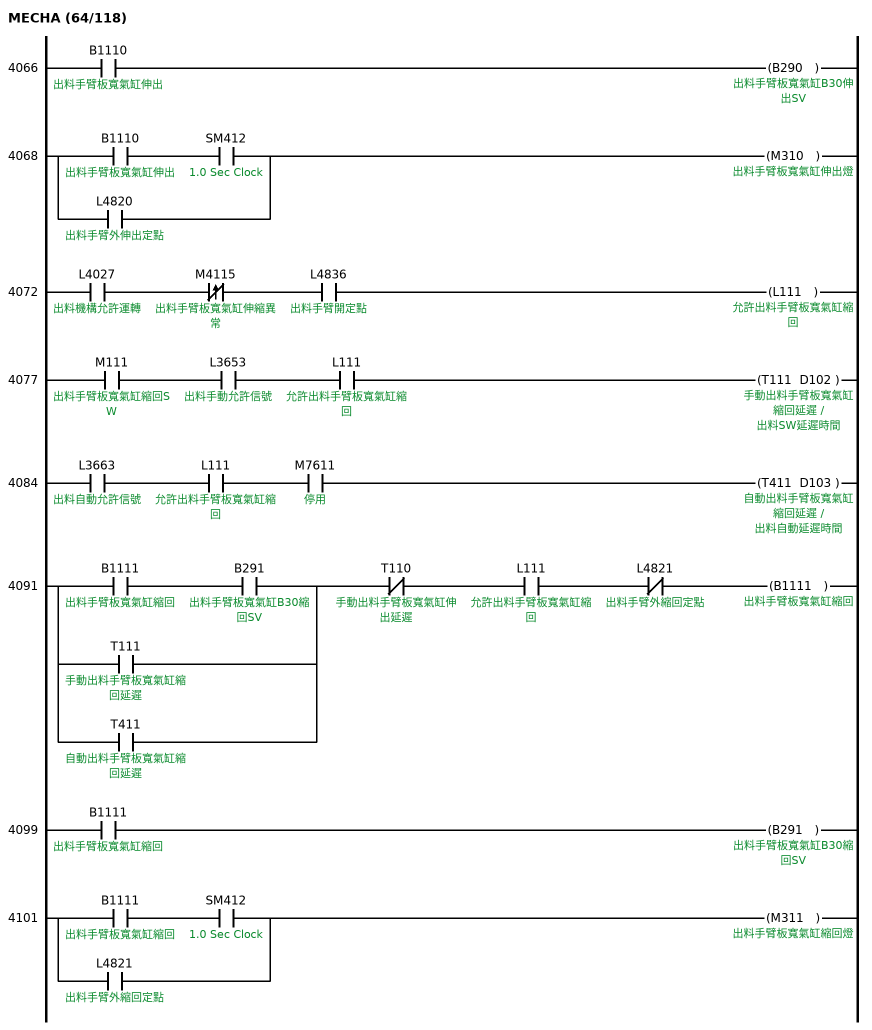
[picture p360: ladder of MECHA, rungs at steps 4066 to 4101]
4066  LD      B1110  ; 出料手臂板寬氣缸伸出
      OUT     B290  ; 出料手臂板寬氣缸B30伸出SV
4068  LD      B1110  ; 出料手臂板寬氣缸伸出
      AND     SM412  ; 1.0 Sec Clock
      OR      L4820  ; 出料手臂外伸出定點
      OUT     M310  ; 出料手臂板寬氣缸伸出燈
4072  LD      L4027  ; 出料機構允許運轉
      ANDPI   M4115  ; 出料手臂板寬氣缸伸縮異常
      AND     L4836  ; 出料手臂開定點
      OUT     L111  ; 允許出料手臂板寬氣缸縮回
4077  LD      M111  ; 出料手臂板寬氣缸縮回SW
      AND     L3653  ; 出料手動允許信號
      AND     L111  ; 允許出料手臂板寬氣缸縮回
      OUT     T111 D102  ; 手動出料手臂板寬氣缸縮回延遲 / 出料SW延遲時間
4084  LD      L3663  ; 出料自動允許信號
      AND     L111  ; 允許出料手臂板寬氣缸縮回
      AND     M7611  ; 停用
      OUT     T411 D103  ; 自動出料手臂板寬氣缸縮回延遲 / 出料自動延遲時間
4091  LD      B1111  ; 出料手臂板寬氣缸縮回
      AND     B291  ; 出料手臂板寬氣缸B30縮回SV
      OR      T111  ; 手動出料手臂板寬氣缸縮回延遲
      OR      T411  ; 自動出料手臂板寬氣缸縮回延遲
      ANI     T110  ; 手動出料手臂板寬氣缸伸出延遲
      AND     L111  ; 允許出料手臂板寬氣缸縮回
      ANI     L4821  ; 出料手臂外縮回定點
      OUT     B1111  ; 出料手臂板寬氣缸縮回
4099  LD      B1111  ; 出料手臂板寬氣缸縮回
      OUT     B291  ; 出料手臂板寬氣缸B30縮回SV
4101  LD      B1111  ; 出料手臂板寬氣缸縮回
      AND     SM412  ; 1.0 Sec Clock
      OR      L4821  ; 出料手臂外縮回定點
      OUT     M311  ; 出料手臂板寬氣缸縮回燈
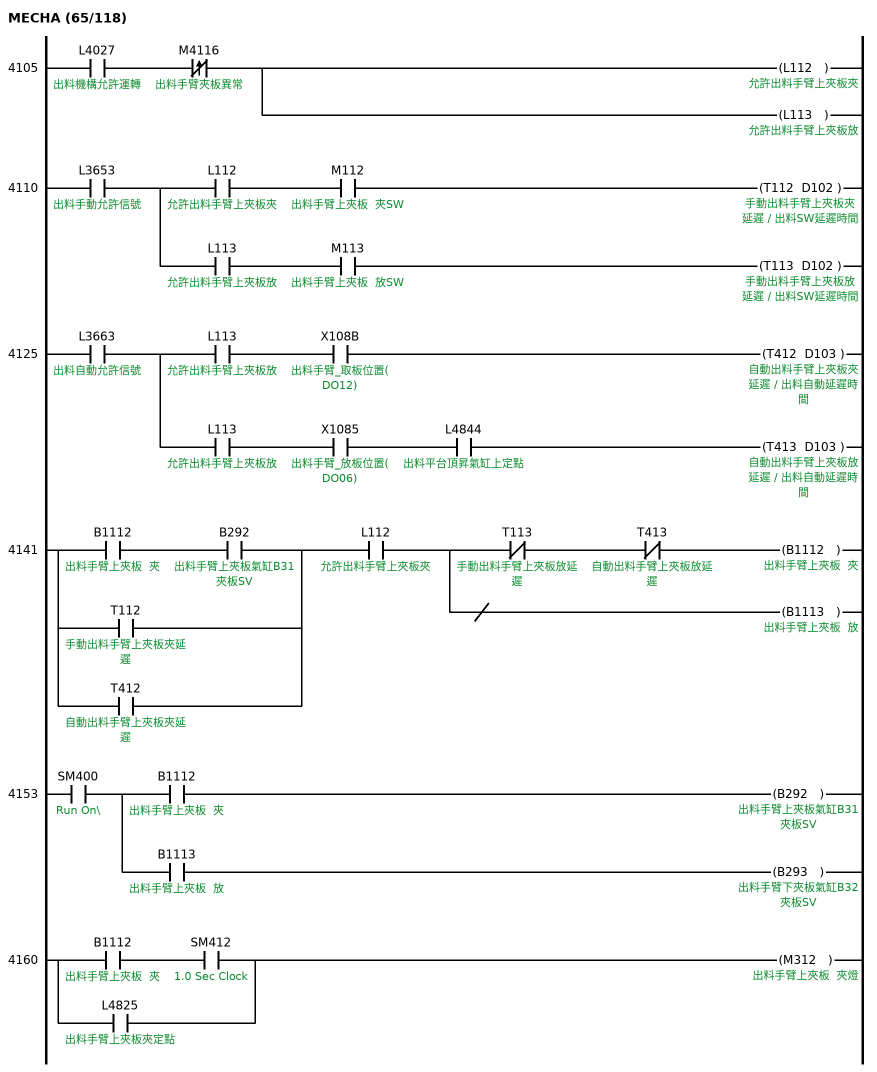
4105  LD      L4027  ; 出料機構允許運轉
      ANDPI   M4116  ; 出料手臂夾板異常
      OUT     L112  ; 允許出料手臂上夾板夾
      OUT     L113  ; 允許出料手臂上夾板放
4110  LD      L3653  ; 出料手動允許信號
      MPS
      AND     L112  ; 允許出料手臂上夾板夾
      AND     M112  ; 出料手臂上夾板  夾SW
      OUT     T112 D102  ; 手動出料手臂上夾板夾延遲 / 出料SW延遲時間
      MPP
      AND     L113  ; 允許出料手臂上夾板放
      AND     M113  ; 出料手臂上夾板  放SW
      OUT     T113 D102  ; 手動出料手臂上夾板放延遲 / 出料SW延遲時間
4125  LD      L3663  ; 出料自動允許信號
      MPS
      AND     L113  ; 允許出料手臂上夾板放
      AND     X108B  ; 出料手臂_取板位置(DO12)
      OUT     T412 D103  ; 自動出料手臂上夾板夾延遲 / 出料自動延遲時間
      MPP
      AND     L113  ; 允許出料手臂上夾板放
      AND     X1085  ; 出料手臂_放板位置(DO06)
      AND     L4844  ; 出料平台頂昇氣缸上定點
      OUT     T413 D103  ; 自動出料手臂上夾板放延遲 / 出料自動延遲時間
4141  LD      B1112  ; 出料手臂上夾板  夾
      AND     B292  ; 出料手臂上夾板氣缸B31夾板SV
      OR      T112  ; 手動出料手臂上夾板夾延遲
      OR      T412  ; 自動出料手臂上夾板夾延遲
      AND     L112  ; 允許出料手臂上夾板夾
      MPS
      ANI     T113  ; 手動出料手臂上夾板放延遲
      ANI     T413  ; 自動出料手臂上夾板放延遲
      OUT     B1112  ; 出料手臂上夾板  夾
      MPP
      INV
      OUT     B1113  ; 出料手臂上夾板  放
4153  LD      SM400  ; Run On\
      MPS
      AND     B1112  ; 出料手臂上夾板  夾
      OUT     B292  ; 出料手臂上夾板氣缸B31夾板SV
      MPP
      AND     B1113  ; 出料手臂上夾板  放
      OUT     B293  ; 出料手臂下夾板氣缸B32夾板SV
4160  LD      B1112  ; 出料手臂上夾板  夾
      AND     SM412  ; 1.0 Sec Clock
      OR      L4825  ; 出料手臂上夾板夾定點
      OUT     M312  ; 出料手臂上夾板  夾燈
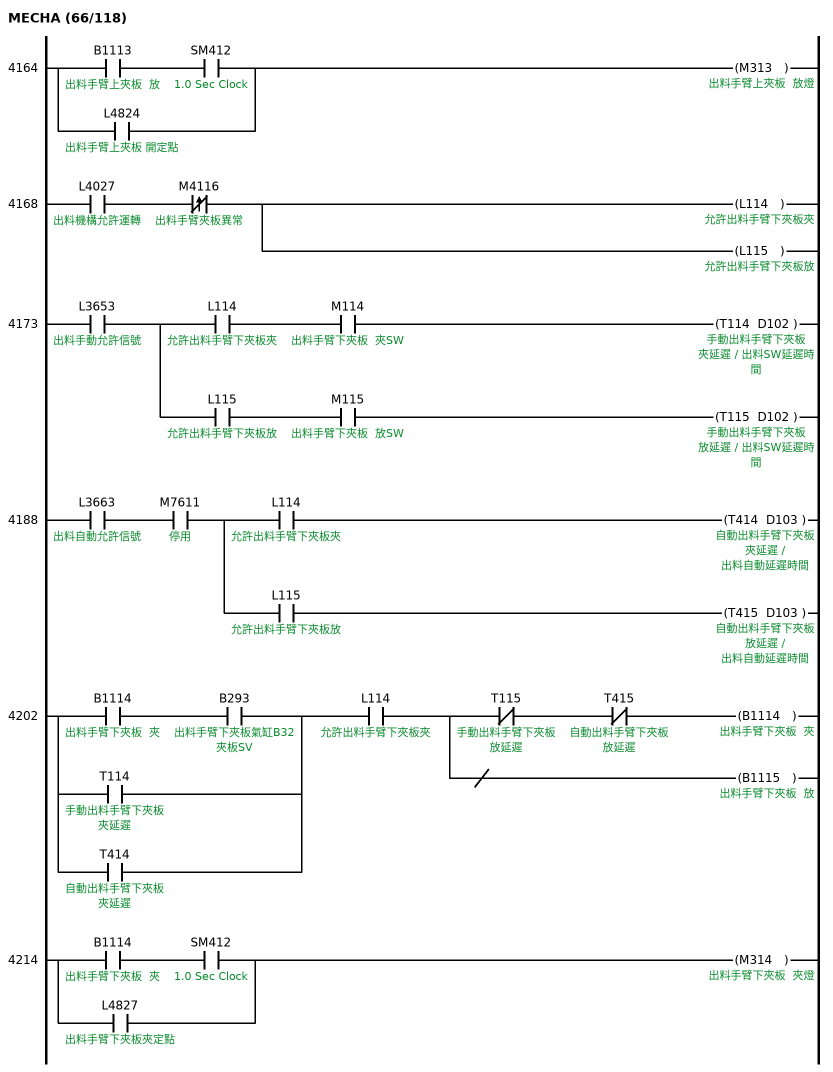
4164  LD      B1113  ; 出料手臂上夾板  放
      AND     SM412  ; 1.0 Sec Clock
      OR      L4824  ; 出料手臂上夾板 開定點
      OUT     M313  ; 出料手臂上夾板  放燈
4168  LD      L4027  ; 出料機構允許運轉
      ANDPI   M4116  ; 出料手臂夾板異常
      OUT     L114  ; 允許出料手臂下夾板夾
      OUT     L115  ; 允許出料手臂下夾板放
4173  LD      L3653  ; 出料手動允許信號
      MPS
      AND     L114  ; 允許出料手臂下夾板夾
      AND     M114  ; 出料手臂下夾板  夾SW
      OUT     T114 D102  ; 手動出料手臂下夾板  夾延遲 / 出料SW延遲時間
      MPP
      AND     L115  ; 允許出料手臂下夾板放
      AND     M115  ; 出料手臂下夾板  放SW
      OUT     T115 D102  ; 手動出料手臂下夾板  放延遲 / 出料SW延遲時間
4188  LD      L3663  ; 出料自動允許信號
      AND     M7611  ; 停用
      MPS
      AND     L114  ; 允許出料手臂下夾板夾
      OUT     T414 D103  ; 自動出料手臂下夾板  夾延遲 / 出料自動延遲時間
      MPP
      AND     L115  ; 允許出料手臂下夾板放
      OUT     T415 D103  ; 自動出料手臂下夾板  放延遲 / 出料自動延遲時間
4202  LD      B1114  ; 出料手臂下夾板  夾
      AND     B293  ; 出料手臂下夾板氣缸B32夾板SV
      OR      T114  ; 手動出料手臂下夾板  夾延遲
      OR      T414  ; 自動出料手臂下夾板  夾延遲
      AND     L114  ; 允許出料手臂下夾板夾
      MPS
      ANI     T115  ; 手動出料手臂下夾板  放延遲
      ANI     T415  ; 自動出料手臂下夾板  放延遲
      OUT     B1114  ; 出料手臂下夾板  夾
      MPP
      INV
      OUT     B1115  ; 出料手臂下夾板  放
4214  LD      B1114  ; 出料手臂下夾板  夾
      AND     SM412  ; 1.0 Sec Clock
      OR      L4827  ; 出料手臂下夾板夾定點
      OUT     M314  ; 出料手臂下夾板  夾燈
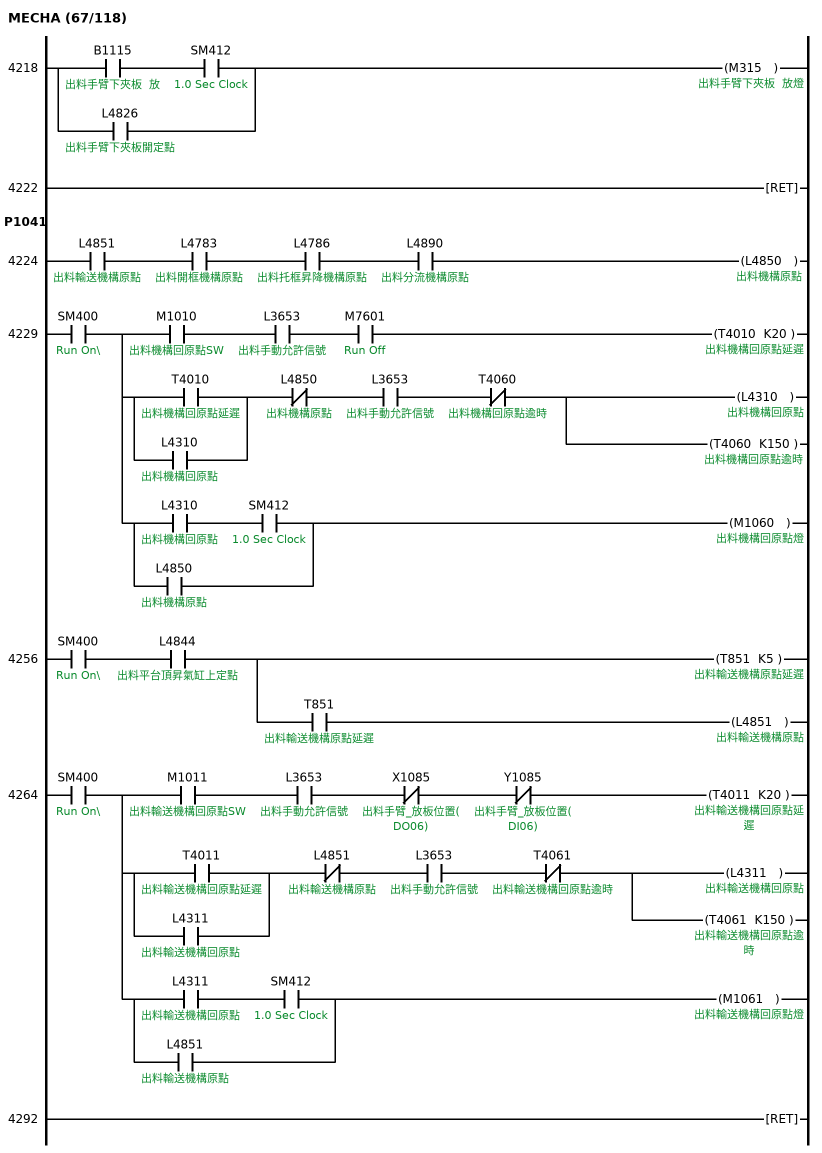
4218  LD      B1115  ; 出料手臂下夾板  放
      AND     SM412  ; 1.0 Sec Clock
      OR      L4826  ; 出料手臂下夾板開定點
      OUT     M315  ; 出料手臂下夾板  放燈
4222  RET
      P1041
4224  LD      L4851  ; 出料輸送機構原點
      AND     L4783  ; 出料開框機構原點
      AND     L4786  ; 出料托框昇降機構原點
      AND     L4890  ; 出料分流機構原點
      OUT     L4850  ; 出料機構原點
4229  LD      SM400  ; Run On\
      MPS
      AND     M1010  ; 出料機構回原點SW
      AND     L3653  ; 出料手動允許信號
      AND     M7601  ; Run Off
      OUT     T4010 K20  ; 出料機構回原點延遲
      MRD
      LD      T4010  ; 出料機構回原點延遲
      OR      L4310  ; 出料機構回原點
      ANB
      ANI     L4850  ; 出料機構原點
      AND     L3653  ; 出料手動允許信號
      ANI     T4060  ; 出料機構回原點逾時
      OUT     L4310  ; 出料機構回原點
      OUT     T4060 K150  ; 出料機構回原點逾時
      MPP
      LD      L4310  ; 出料機構回原點
      AND     SM412  ; 1.0 Sec Clock
      OR      L4850  ; 出料機構原點
      ANB
      OUT     M1060  ; 出料機構回原點燈
4256  LD      SM400  ; Run On\
      AND     L4844  ; 出料平台頂昇氣缸上定點
      OUT     T851 K5  ; 出料輸送機構原點延遲
      AND     T851  ; 出料輸送機構原點延遲
      OUT     L4851  ; 出料輸送機構原點
4264  LD      SM400  ; Run On\
      MPS
      AND     M1011  ; 出料輸送機構回原點SW
      AND     L3653  ; 出料手動允許信號
      ANI     X1085  ; 出料手臂_放板位置(DO06)
      ANI     Y1085  ; 出料手臂_放板位置(DI06)
      OUT     T4011 K20  ; 出料輸送機構回原點延遲
      MRD
      LD      T4011  ; 出料輸送機構回原點延遲
      OR      L4311  ; 出料輸送機構回原點
      ANB
      ANI     L4851  ; 出料輸送機構原點
      AND     L3653  ; 出料手動允許信號
      ANI     T4061  ; 出料輸送機構回原點逾時
      OUT     L4311  ; 出料輸送機構回原點
      OUT     T4061 K150  ; 出料輸送機構回原點逾時
      MPP
      LD      L4311  ; 出料輸送機構回原點
      AND     SM412  ; 1.0 Sec Clock
      OR      L4851  ; 出料輸送機構原點
      ANB
      OUT     M1061  ; 出料輸送機構回原點燈
4292  RET
; 出料回流下導框機構
      P1050
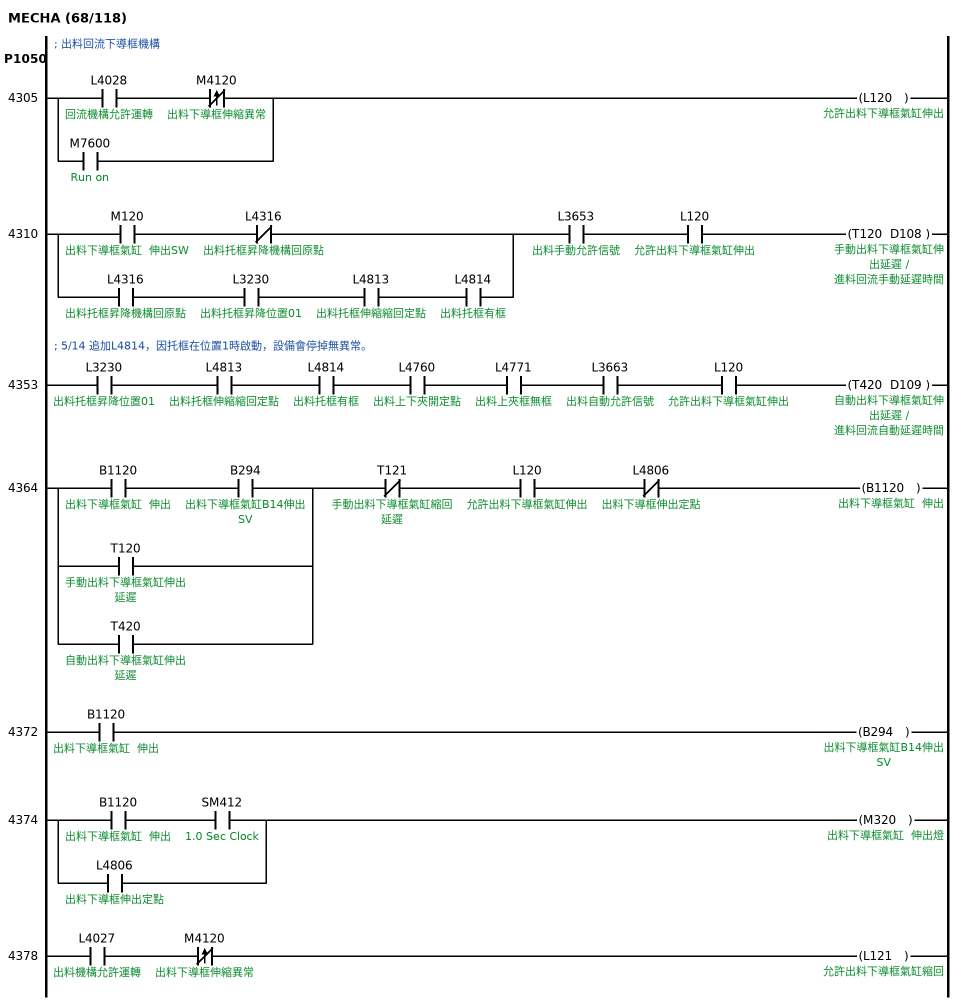
4305  LD      L4028  ; 回流機構允許運轉
      ANDPI   M4120  ; 出料下導框伸縮異常
      OR      M7600  ; Run on
      OUT     L120  ; 允許出料下導框氣缸伸出
4310  LD      M120  ; 出料下導框氣缸  伸出SW
      ANI     L4316  ; 出料托框昇降機構回原點
      LD      L4316  ; 出料托框昇降機構回原點
      AND     L3230  ; 出料托框昇降位置01
      AND     L4813  ; 出料托框伸縮縮回定點
      AND     L4814  ; 出料托框有框
      ORB
      AND     L3653  ; 出料手動允許信號
      AND     L120  ; 允許出料下導框氣缸伸出
      OUT     T120 D108  ; 手動出料下導框氣缸伸出延遲 / 進料回流手動延遲時間
; 5/14 追加L4814，因托框在位置1時啟動，設備會停掉無異常。
4353  LD      L3230  ; 出料托框昇降位置01
      AND     L4813  ; 出料托框伸縮縮回定點
      AND     L4814  ; 出料托框有框
      AND     L4760  ; 出料上下夾開定點
      AND     L4771  ; 出料上夾框無框
      AND     L3663  ; 出料自動允許信號
      AND     L120  ; 允許出料下導框氣缸伸出
      OUT     T420 D109  ; 自動出料下導框氣缸伸出延遲 / 進料回流自動延遲時間
4364  LD      B1120  ; 出料下導框氣缸  伸出
      AND     B294  ; 出料下導框氣缸B14伸出SV
      OR      T120  ; 手動出料下導框氣缸伸出延遲
      OR      T420  ; 自動出料下導框氣缸伸出延遲
      ANI     T121  ; 手動出料下導框氣缸縮回延遲
      AND     L120  ; 允許出料下導框氣缸伸出
      ANI     L4806  ; 出料下導框伸出定點
      OUT     B1120  ; 出料下導框氣缸  伸出
4372  LD      B1120  ; 出料下導框氣缸  伸出
      OUT     B294  ; 出料下導框氣缸B14伸出SV
4374  LD      B1120  ; 出料下導框氣缸  伸出
      AND     SM412  ; 1.0 Sec Clock
      OR      L4806  ; 出料下導框伸出定點
      OUT     M320  ; 出料下導框氣缸  伸出燈
4378  LD      L4027  ; 出料機構允許運轉
      ANDPI   M4120  ; 出料下導框伸縮異常
      OUT     L121  ; 允許出料下導框氣缸縮回
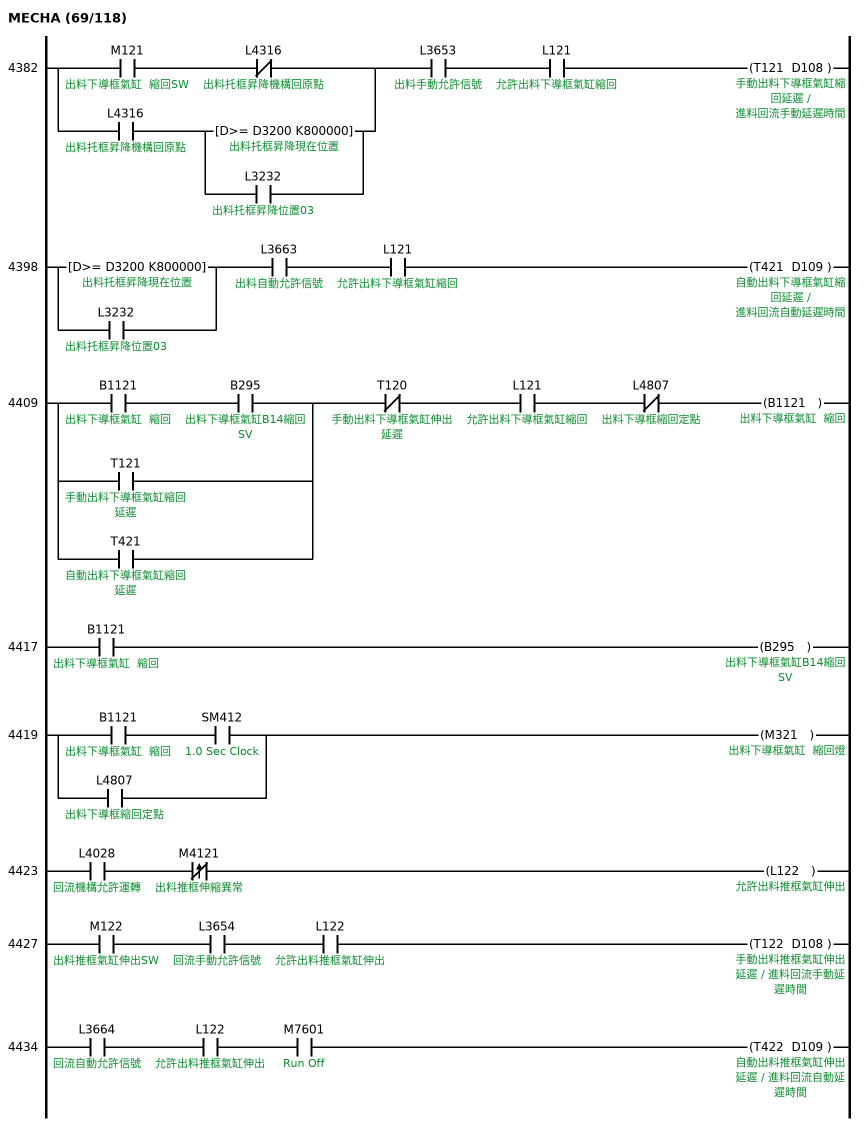
4382  LD      M121  ; 出料下導框氣缸  縮回SW
      ANI     L4316  ; 出料托框昇降機構回原點
      LD      L4316  ; 出料托框昇降機構回原點
      LDD>=   D3200 K800000  ; 出料托框昇降現在位置
      OR      L3232  ; 出料托框昇降位置03
      ANB
      ORB
      AND     L3653  ; 出料手動允許信號
      AND     L121  ; 允許出料下導框氣缸縮回
      OUT     T121 D108  ; 手動出料下導框氣缸縮回延遲 / 進料回流手動延遲時間
4398  LDD>=   D3200 K800000  ; 出料托框昇降現在位置
      OR      L3232  ; 出料托框昇降位置03
      AND     L3663  ; 出料自動允許信號
      AND     L121  ; 允許出料下導框氣缸縮回
      OUT     T421 D109  ; 自動出料下導框氣缸縮回延遲 / 進料回流自動延遲時間
4409  LD      B1121  ; 出料下導框氣缸  縮回
      AND     B295  ; 出料下導框氣缸B14縮回SV
      OR      T121  ; 手動出料下導框氣缸縮回延遲
      OR      T421  ; 自動出料下導框氣缸縮回延遲
      ANI     T120  ; 手動出料下導框氣缸伸出延遲
      AND     L121  ; 允許出料下導框氣缸縮回
      ANI     L4807  ; 出料下導框縮回定點
      OUT     B1121  ; 出料下導框氣缸  縮回
4417  LD      B1121  ; 出料下導框氣缸  縮回
      OUT     B295  ; 出料下導框氣缸B14縮回SV
4419  LD      B1121  ; 出料下導框氣缸  縮回
      AND     SM412  ; 1.0 Sec Clock
      OR      L4807  ; 出料下導框縮回定點
      OUT     M321  ; 出料下導框氣缸  縮回燈
4423  LD      L4028  ; 回流機構允許運轉
      ANDPI   M4121  ; 出料推框伸縮異常
      OUT     L122  ; 允許出料推框氣缸伸出
4427  LD      M122  ; 出料推框氣缸伸出SW
      AND     L3654  ; 回流手動允許信號
      AND     L122  ; 允許出料推框氣缸伸出
      OUT     T122 D108  ; 手動出料推框氣缸伸出延遲 / 進料回流手動延遲時間
4434  LD      L3664  ; 回流自動允許信號
      AND     L122  ; 允許出料推框氣缸伸出
      AND     M7601  ; Run Off
      OUT     T422 D109  ; 自動出料推框氣缸伸出延遲 / 進料回流自動延遲時間
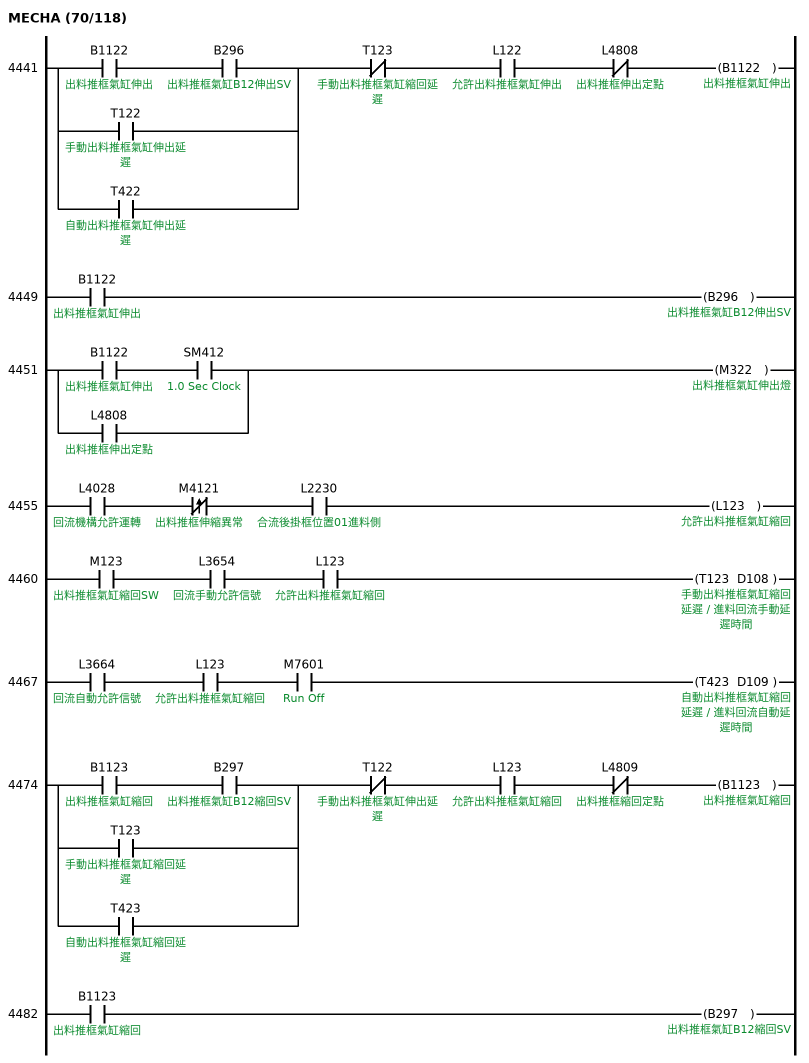
4441  LD      B1122  ; 出料推框氣缸伸出
      AND     B296  ; 出料推框氣缸B12伸出SV
      OR      T122  ; 手動出料推框氣缸伸出延遲
      OR      T422  ; 自動出料推框氣缸伸出延遲
      ANI     T123  ; 手動出料推框氣缸縮回延遲
      AND     L122  ; 允許出料推框氣缸伸出
      ANI     L4808  ; 出料推框伸出定點
      OUT     B1122  ; 出料推框氣缸伸出
4449  LD      B1122  ; 出料推框氣缸伸出
      OUT     B296  ; 出料推框氣缸B12伸出SV
4451  LD      B1122  ; 出料推框氣缸伸出
      AND     SM412  ; 1.0 Sec Clock
      OR      L4808  ; 出料推框伸出定點
      OUT     M322  ; 出料推框氣缸伸出燈
4455  LD      L4028  ; 回流機構允許運轉
      ANDPI   M4121  ; 出料推框伸縮異常
      AND     L2230  ; 合流後掛框位置01進料側
      OUT     L123  ; 允許出料推框氣缸縮回
4460  LD      M123  ; 出料推框氣缸縮回SW
      AND     L3654  ; 回流手動允許信號
      AND     L123  ; 允許出料推框氣缸縮回
      OUT     T123 D108  ; 手動出料推框氣缸縮回延遲 / 進料回流手動延遲時間
4467  LD      L3664  ; 回流自動允許信號
      AND     L123  ; 允許出料推框氣缸縮回
      AND     M7601  ; Run Off
      OUT     T423 D109  ; 自動出料推框氣缸縮回延遲 / 進料回流自動延遲時間
4474  LD      B1123  ; 出料推框氣缸縮回
      AND     B297  ; 出料推框氣缸B12縮回SV
      OR      T123  ; 手動出料推框氣缸縮回延遲
      OR      T423  ; 自動出料推框氣缸縮回延遲
      ANI     T122  ; 手動出料推框氣缸伸出延遲
      AND     L123  ; 允許出料推框氣缸縮回
      ANI     L4809  ; 出料推框縮回定點
      OUT     B1123  ; 出料推框氣缸縮回
4482  LD      B1123  ; 出料推框氣缸縮回
      OUT     B297  ; 出料推框氣缸B12縮回SV
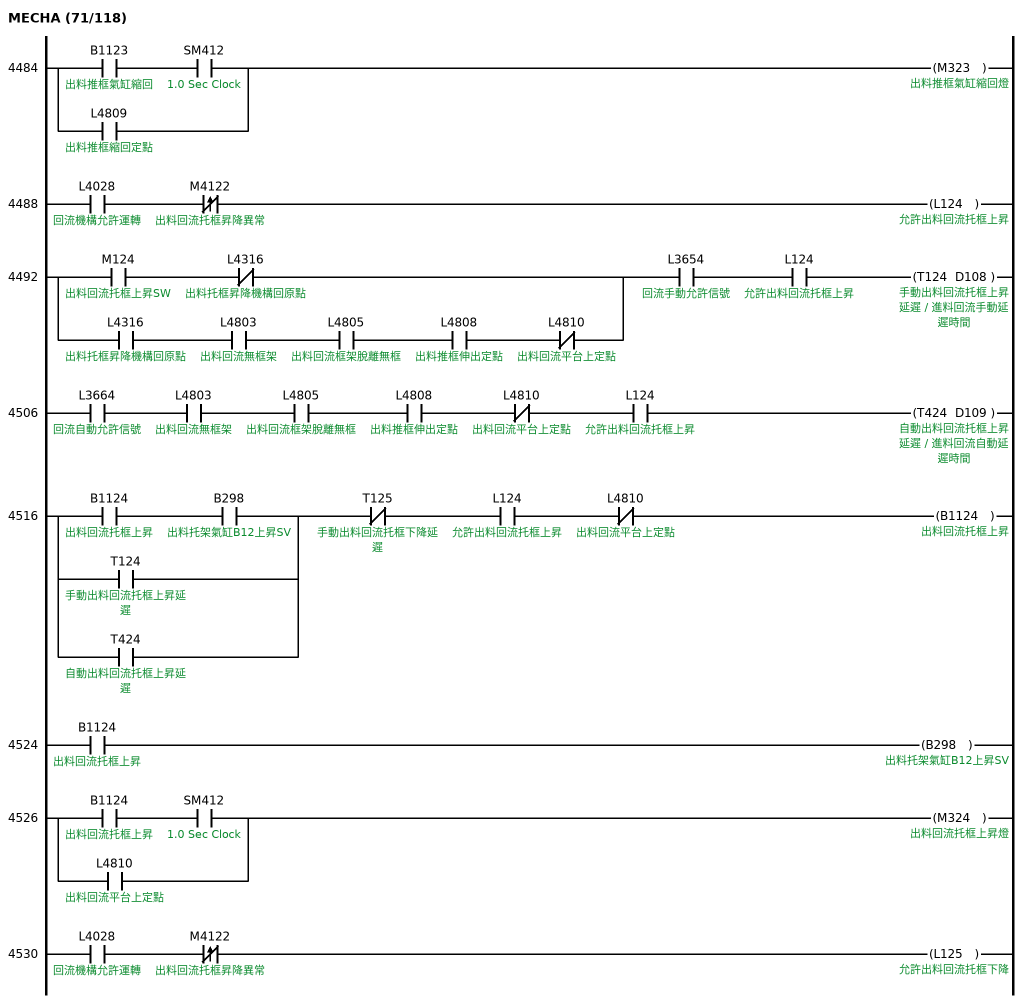
4484  LD      B1123  ; 出料推框氣缸縮回
      AND     SM412  ; 1.0 Sec Clock
      OR      L4809  ; 出料推框縮回定點
      OUT     M323  ; 出料推框氣缸縮回燈
4488  LD      L4028  ; 回流機構允許運轉
      ANDPI   M4122  ; 出料回流托框昇降異常
      OUT     L124  ; 允許出料回流托框上昇
4492  LD      M124  ; 出料回流托框上昇SW
      ANI     L4316  ; 出料托框昇降機構回原點
      LD      L4316  ; 出料托框昇降機構回原點
      AND     L4803  ; 出料回流無框架
      AND     L4805  ; 出料回流框架脫離無框
      AND     L4808  ; 出料推框伸出定點
      ANI     L4810  ; 出料回流平台上定點
      ORB
      AND     L3654  ; 回流手動允許信號
      AND     L124  ; 允許出料回流托框上昇
      OUT     T124 D108  ; 手動出料回流托框上昇延遲 / 進料回流手動延遲時間
4506  LD      L3664  ; 回流自動允許信號
      AND     L4803  ; 出料回流無框架
      AND     L4805  ; 出料回流框架脫離無框
      AND     L4808  ; 出料推框伸出定點
      ANI     L4810  ; 出料回流平台上定點
      AND     L124  ; 允許出料回流托框上昇
      OUT     T424 D109  ; 自動出料回流托框上昇延遲 / 進料回流自動延遲時間
4516  LD      B1124  ; 出料回流托框上昇
      AND     B298  ; 出料托架氣缸B12上昇SV
      OR      T124  ; 手動出料回流托框上昇延遲
      OR      T424  ; 自動出料回流托框上昇延遲
      ANI     T125  ; 手動出料回流托框下降延遲
      AND     L124  ; 允許出料回流托框上昇
      ANI     L4810  ; 出料回流平台上定點
      OUT     B1124  ; 出料回流托框上昇
4524  LD      B1124  ; 出料回流托框上昇
      OUT     B298  ; 出料托架氣缸B12上昇SV
4526  LD      B1124  ; 出料回流托框上昇
      AND     SM412  ; 1.0 Sec Clock
      OR      L4810  ; 出料回流平台上定點
      OUT     M324  ; 出料回流托框上昇燈
4530  LD      L4028  ; 回流機構允許運轉
      ANDPI   M4122  ; 出料回流托框昇降異常
      OUT     L125  ; 允許出料回流托框下降
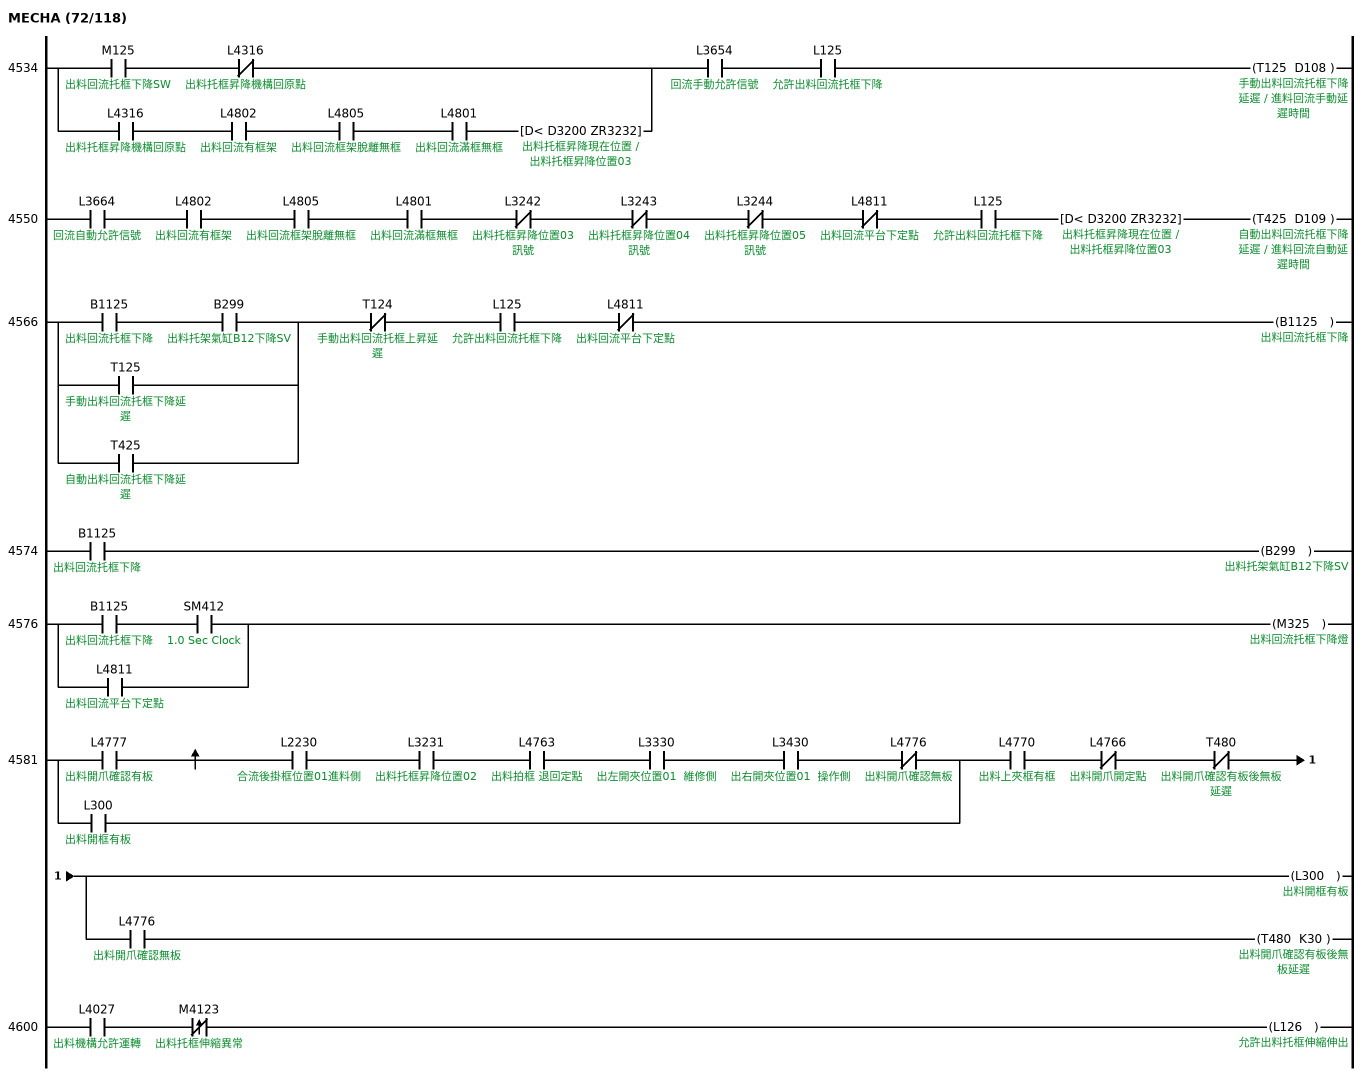
4534  LD      M125  ; 出料回流托框下降SW
      ANI     L4316  ; 出料托框昇降機構回原點
      LD      L4316  ; 出料托框昇降機構回原點
      AND     L4802  ; 出料回流有框架
      AND     L4805  ; 出料回流框架脫離無框
      AND     L4801  ; 出料回流滿框無框
      ANDD<   D3200 ZR3232  ; 出料托框昇降現在位置 / 出料托框昇降位置03
      ORB
      AND     L3654  ; 回流手動允許信號
      AND     L125  ; 允許出料回流托框下降
      OUT     T125 D108  ; 手動出料回流托框下降延遲 / 進料回流手動延遲時間
4550  LD      L3664  ; 回流自動允許信號
      AND     L4802  ; 出料回流有框架
      AND     L4805  ; 出料回流框架脫離無框
      AND     L4801  ; 出料回流滿框無框
      ANI     L3242  ; 出料托框昇降位置03 訊號
      ANI     L3243  ; 出料托框昇降位置04 訊號
      ANI     L3244  ; 出料托框昇降位置05 訊號
      ANI     L4811  ; 出料回流平台下定點
      AND     L125  ; 允許出料回流托框下降
      ANDD<   D3200 ZR3232  ; 出料托框昇降現在位置 / 出料托框昇降位置03
      OUT     T425 D109  ; 自動出料回流托框下降延遲 / 進料回流自動延遲時間
4566  LD      B1125  ; 出料回流托框下降
      AND     B299  ; 出料托架氣缸B12下降SV
      OR      T125  ; 手動出料回流托框下降延遲
      OR      T425  ; 自動出料回流托框下降延遲
      ANI     T124  ; 手動出料回流托框上昇延遲
      AND     L125  ; 允許出料回流托框下降
      ANI     L4811  ; 出料回流平台下定點
      OUT     B1125  ; 出料回流托框下降
4574  LD      B1125  ; 出料回流托框下降
      OUT     B299  ; 出料托架氣缸B12下降SV
4576  LD      B1125  ; 出料回流托框下降
      AND     SM412  ; 1.0 Sec Clock
      OR      L4811  ; 出料回流平台下定點
      OUT     M325  ; 出料回流托框下降燈
4581  LD      L4777  ; 出料開爪確認有板
      MEP
      AND     L2230  ; 合流後掛框位置01進料側
      AND     L3231  ; 出料托框昇降位置02
      AND     L4763  ; 出料拍框 退回定點
      AND     L3330  ; 出左開夾位置01  維修側
      AND     L3430  ; 出右開夾位置01  操作側
      ANI     L4776  ; 出料開爪確認無板
      OR      L300  ; 出料開框有板
      AND     L4770  ; 出料上夾框有框
      ANI     L4766  ; 出料開爪開定點
      ANI     T480  ; 出料開爪確認有板後無板延遲
      OUT     L300  ; 出料開框有板
      AND     L4776  ; 出料開爪確認無板
      OUT     T480 K30  ; 出料開爪確認有板後無板延遲
4600  LD      L4027  ; 出料機構允許運轉
      ANDPI   M4123  ; 出料托框伸縮異常
      OUT     L126  ; 允許出料托框伸縮伸出
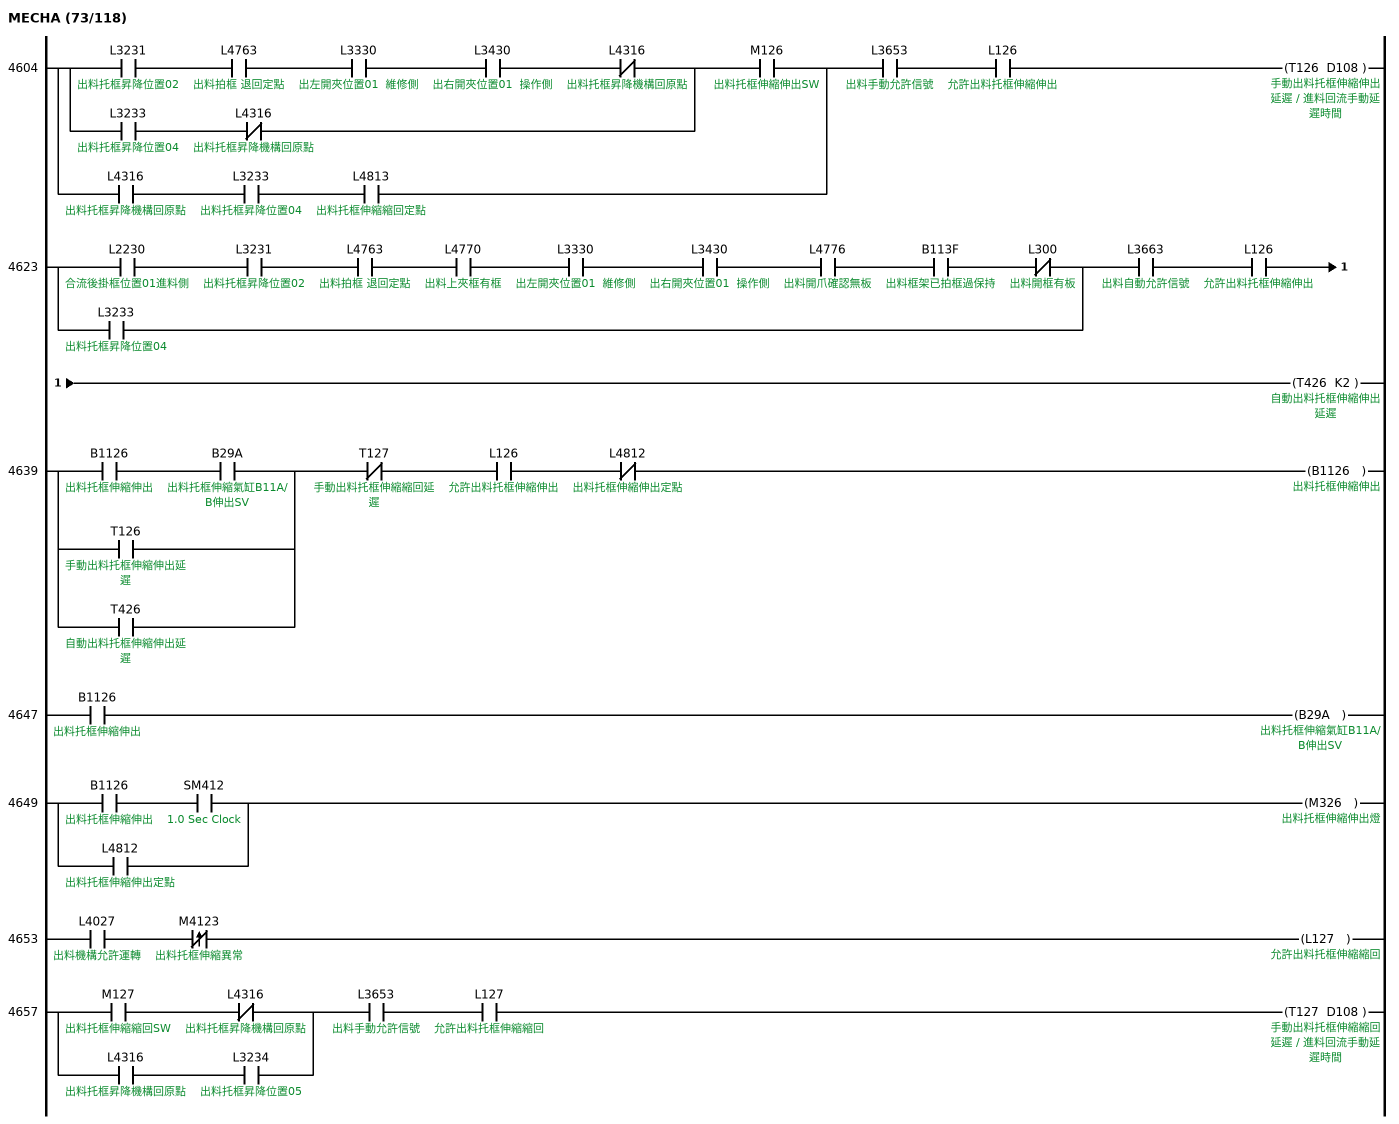
4604  LD      L3231  ; 出料托框昇降位置02
      AND     L4763  ; 出料拍框 退回定點
      AND     L3330  ; 出左開夾位置01  維修側
      AND     L3430  ; 出右開夾位置01  操作側
      ANI     L4316  ; 出料托框昇降機構回原點
      LD      L3233  ; 出料托框昇降位置04
      ANI     L4316  ; 出料托框昇降機構回原點
      ORB
      AND     M126  ; 出料托框伸縮伸出SW
      LD      L4316  ; 出料托框昇降機構回原點
      AND     L3233  ; 出料托框昇降位置04
      AND     L4813  ; 出料托框伸縮縮回定點
      ORB
      AND     L3653  ; 出料手動允許信號
      AND     L126  ; 允許出料托框伸縮伸出
      OUT     T126 D108  ; 手動出料托框伸縮伸出延遲 / 進料回流手動延遲時間
4623  LD      L2230  ; 合流後掛框位置01進料側
      AND     L3231  ; 出料托框昇降位置02
      AND     L4763  ; 出料拍框 退回定點
      AND     L4770  ; 出料上夾框有框
      AND     L3330  ; 出左開夾位置01  維修側
      AND     L3430  ; 出右開夾位置01  操作側
      AND     L4776  ; 出料開爪確認無板
      AND     B113F  ; 出料框架已拍框過保持
      ANI     L300  ; 出料開框有板
      OR      L3233  ; 出料托框昇降位置04
      AND     L3663  ; 出料自動允許信號
      AND     L126  ; 允許出料托框伸縮伸出
      OUT     T426 K2  ; 自動出料托框伸縮伸出延遲
4639  LD      B1126  ; 出料托框伸縮伸出
      AND     B29A  ; 出料托框伸縮氣缸B11A/B伸出SV
      OR      T126  ; 手動出料托框伸縮伸出延遲
      OR      T426  ; 自動出料托框伸縮伸出延遲
      ANI     T127  ; 手動出料托框伸縮縮回延遲
      AND     L126  ; 允許出料托框伸縮伸出
      ANI     L4812  ; 出料托框伸縮伸出定點
      OUT     B1126  ; 出料托框伸縮伸出
4647  LD      B1126  ; 出料托框伸縮伸出
      OUT     B29A  ; 出料托框伸縮氣缸B11A/B伸出SV
4649  LD      B1126  ; 出料托框伸縮伸出
      AND     SM412  ; 1.0 Sec Clock
      OR      L4812  ; 出料托框伸縮伸出定點
      OUT     M326  ; 出料托框伸縮伸出燈
4653  LD      L4027  ; 出料機構允許運轉
      ANDPI   M4123  ; 出料托框伸縮異常
      OUT     L127  ; 允許出料托框伸縮縮回
4657  LD      M127  ; 出料托框伸縮縮回SW
      ANI     L4316  ; 出料托框昇降機構回原點
      LD      L4316  ; 出料托框昇降機構回原點
      AND     L3234  ; 出料托框昇降位置05
      ORB
      AND     L3653  ; 出料手動允許信號
      AND     L127  ; 允許出料托框伸縮縮回
      OUT     T127 D108  ; 手動出料托框伸縮縮回延遲 / 進料回流手動延遲時間
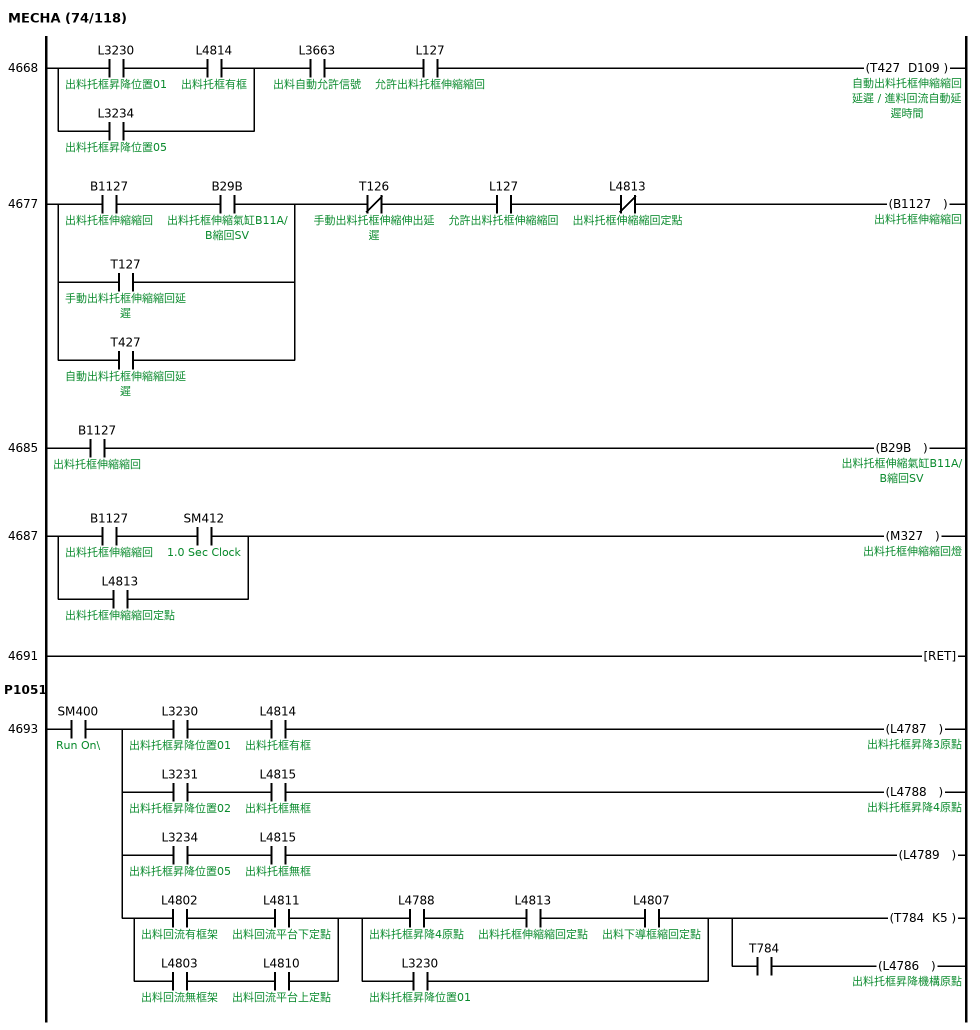
4668  LD      L3230  ; 出料托框昇降位置01
      AND     L4814  ; 出料托框有框
      OR      L3234  ; 出料托框昇降位置05
      AND     L3663  ; 出料自動允許信號
      AND     L127  ; 允許出料托框伸縮縮回
      OUT     T427 D109  ; 自動出料托框伸縮縮回延遲 / 進料回流自動延遲時間
4677  LD      B1127  ; 出料托框伸縮縮回
      AND     B29B  ; 出料托框伸縮氣缸B11A/B縮回SV
      OR      T127  ; 手動出料托框伸縮縮回延遲
      OR      T427  ; 自動出料托框伸縮縮回延遲
      ANI     T126  ; 手動出料托框伸縮伸出延遲
      AND     L127  ; 允許出料托框伸縮縮回
      ANI     L4813  ; 出料托框伸縮縮回定點
      OUT     B1127  ; 出料托框伸縮縮回
4685  LD      B1127  ; 出料托框伸縮縮回
      OUT     B29B  ; 出料托框伸縮氣缸B11A/B縮回SV
4687  LD      B1127  ; 出料托框伸縮縮回
      AND     SM412  ; 1.0 Sec Clock
      OR      L4813  ; 出料托框伸縮縮回定點
      OUT     M327  ; 出料托框伸縮縮回燈
4691  RET
      P1051
4693  LD      SM400  ; Run On\
      MPS
      AND     L3230  ; 出料托框昇降位置01
      AND     L4814  ; 出料托框有框
      OUT     L4787  ; 出料托框昇降3原點
      MRD
      AND     L3231  ; 出料托框昇降位置02
      AND     L4815  ; 出料托框無框
      OUT     L4788  ; 出料托框昇降4原點
      MRD
      AND     L3234  ; 出料托框昇降位置05
      AND     L4815  ; 出料托框無框
      OUT     L4789
      MPP
      LD      L4802  ; 出料回流有框架
      AND     L4811  ; 出料回流平台下定點
      LD      L4803  ; 出料回流無框架
      AND     L4810  ; 出料回流平台上定點
      ORB
      ANB
      LD      L4788  ; 出料托框昇降4原點
      AND     L4813  ; 出料托框伸縮縮回定點
      AND     L4807  ; 出料下導框縮回定點
      OR      L3230  ; 出料托框昇降位置01
      ANB
      OUT     T784 K5
      AND     T784
      OUT     L4786  ; 出料托框昇降機構原點
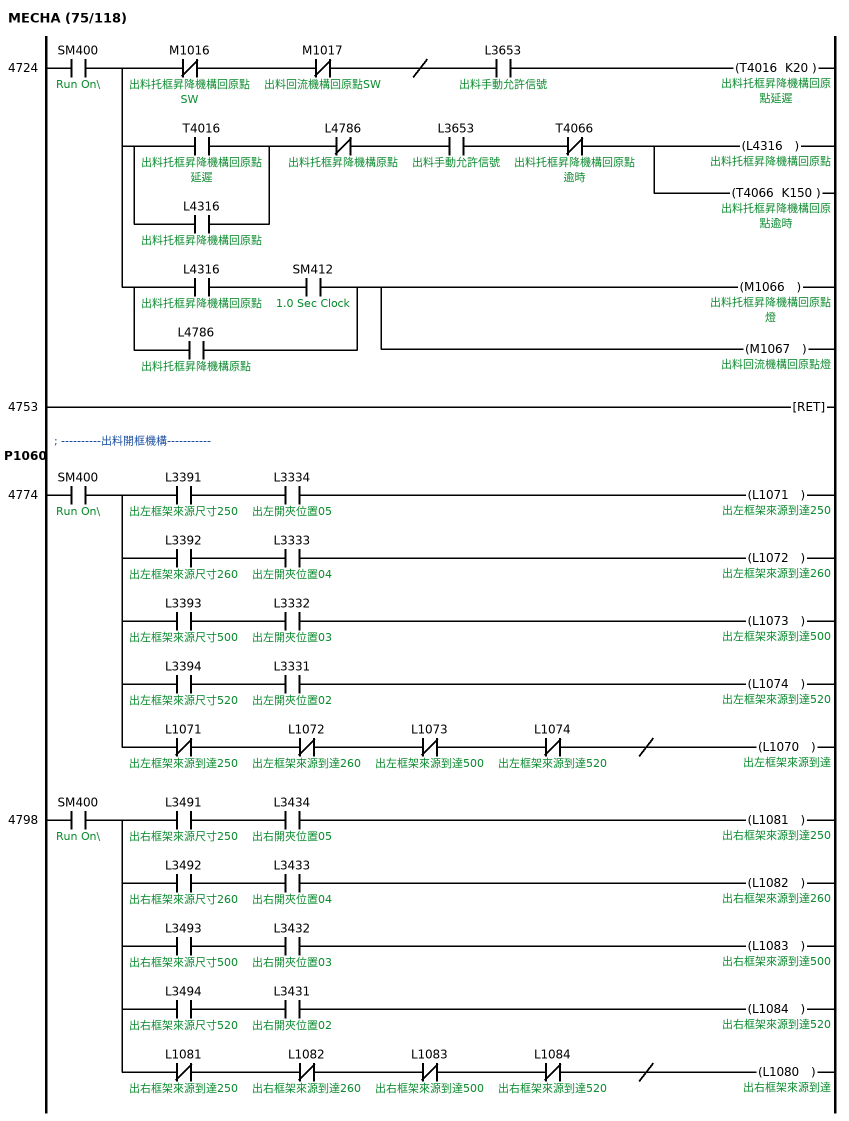
4724  LD      SM400  ; Run On\
      MPS
      ANI     M1016  ; 出料托框昇降機構回原點SW
      ANI     M1017  ; 出料回流機構回原點SW
      INV
      AND     L3653  ; 出料手動允許信號
      OUT     T4016 K20  ; 出料托框昇降機構回原點延遲
      MRD
      LD      T4016  ; 出料托框昇降機構回原點延遲
      OR      L4316  ; 出料托框昇降機構回原點
      ANB
      ANI     L4786  ; 出料托框昇降機構原點
      AND     L3653  ; 出料手動允許信號
      ANI     T4066  ; 出料托框昇降機構回原點逾時
      OUT     L4316  ; 出料托框昇降機構回原點
      OUT     T4066 K150  ; 出料托框昇降機構回原點逾時
      MPP
      LD      L4316  ; 出料托框昇降機構回原點
      AND     SM412  ; 1.0 Sec Clock
      OR      L4786  ; 出料托框昇降機構原點
      ANB
      OUT     M1066  ; 出料托框昇降機構回原點燈
      OUT     M1067  ; 出料回流機構回原點燈
4753  RET
; ----------出料開框機構-----------
      P1060
4774  LD      SM400  ; Run On\
      MPS
      AND     L3391  ; 出左框架來源尺寸250
      AND     L3334  ; 出左開夾位置05
      OUT     L1071  ; 出左框架來源到達250
      MRD
      AND     L3392  ; 出左框架來源尺寸260
      AND     L3333  ; 出左開夾位置04
      OUT     L1072  ; 出左框架來源到達260
      MRD
      AND     L3393  ; 出左框架來源尺寸500
      AND     L3332  ; 出左開夾位置03
      OUT     L1073  ; 出左框架來源到達500
      MRD
      AND     L3394  ; 出左框架來源尺寸520
      AND     L3331  ; 出左開夾位置02
      OUT     L1074  ; 出左框架來源到達520
      MPP
      ANI     L1071  ; 出左框架來源到達250
      ANI     L1072  ; 出左框架來源到達260
      ANI     L1073  ; 出左框架來源到達500
      ANI     L1074  ; 出左框架來源到達520
      INV
      OUT     L1070  ; 出左框架來源到達
4798  LD      SM400  ; Run On\
      MPS
      AND     L3491  ; 出右框架來源尺寸250
      AND     L3434  ; 出右開夾位置05
      OUT     L1081  ; 出右框架來源到達250
      MRD
      AND     L3492  ; 出右框架來源尺寸260
      AND     L3433  ; 出右開夾位置04
      OUT     L1082  ; 出右框架來源到達260
      MRD
      AND     L3493  ; 出右框架來源尺寸500
      AND     L3432  ; 出右開夾位置03
      OUT     L1083  ; 出右框架來源到達500
      MRD
      AND     L3494  ; 出右框架來源尺寸520
      AND     L3431  ; 出右開夾位置02
      OUT     L1084  ; 出右框架來源到達520
      MPP
      ANI     L1081  ; 出右框架來源到達250
      ANI     L1082  ; 出右框架來源到達260
      ANI     L1083  ; 出右框架來源到達500
      ANI     L1084  ; 出右框架來源到達520
      INV
      OUT     L1080  ; 出右框架來源到達
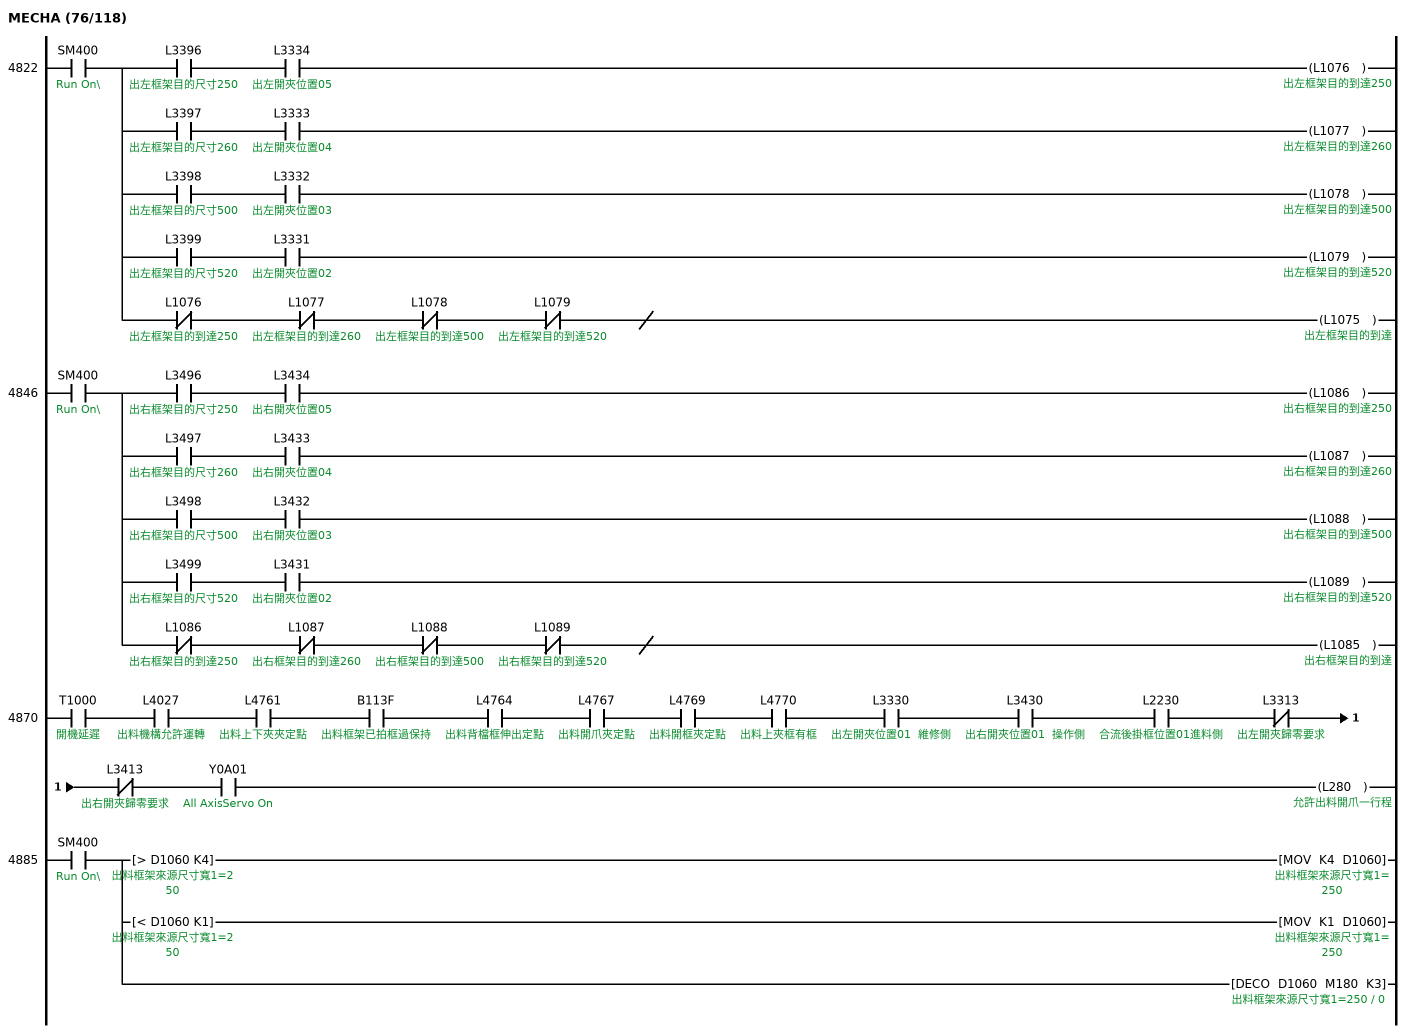
4822  LD      SM400  ; Run On\
      MPS
      AND     L3396  ; 出左框架目的尺寸250
      AND     L3334  ; 出左開夾位置05
      OUT     L1076  ; 出左框架目的到達250
      MRD
      AND     L3397  ; 出左框架目的尺寸260
      AND     L3333  ; 出左開夾位置04
      OUT     L1077  ; 出左框架目的到達260
      MRD
      AND     L3398  ; 出左框架目的尺寸500
      AND     L3332  ; 出左開夾位置03
      OUT     L1078  ; 出左框架目的到達500
      MRD
      AND     L3399  ; 出左框架目的尺寸520
      AND     L3331  ; 出左開夾位置02
      OUT     L1079  ; 出左框架目的到達520
      MPP
      ANI     L1076  ; 出左框架目的到達250
      ANI     L1077  ; 出左框架目的到達260
      ANI     L1078  ; 出左框架目的到達500
      ANI     L1079  ; 出左框架目的到達520
      INV
      OUT     L1075  ; 出左框架目的到達
4846  LD      SM400  ; Run On\
      MPS
      AND     L3496  ; 出右框架目的尺寸250
      AND     L3434  ; 出右開夾位置05
      OUT     L1086  ; 出右框架目的到達250
      MRD
      AND     L3497  ; 出右框架目的尺寸260
      AND     L3433  ; 出右開夾位置04
      OUT     L1087  ; 出右框架目的到達260
      MRD
      AND     L3498  ; 出右框架目的尺寸500
      AND     L3432  ; 出右開夾位置03
      OUT     L1088  ; 出右框架目的到達500
      MRD
      AND     L3499  ; 出右框架目的尺寸520
      AND     L3431  ; 出右開夾位置02
      OUT     L1089  ; 出右框架目的到達520
      MPP
      ANI     L1086  ; 出右框架目的到達250
      ANI     L1087  ; 出右框架目的到達260
      ANI     L1088  ; 出右框架目的到達500
      ANI     L1089  ; 出右框架目的到達520
      INV
      OUT     L1085  ; 出右框架目的到達
4870  LD      T1000  ; 開機延遲
      AND     L4027  ; 出料機構允許運轉
      AND     L4761  ; 出料上下夾夾定點
      AND     B113F  ; 出料框架已拍框過保持
      AND     L4764  ; 出料背檔框伸出定點
      AND     L4767  ; 出料開爪夾定點
      AND     L4769  ; 出料開框夾定點
      AND     L4770  ; 出料上夾框有框
      AND     L3330  ; 出左開夾位置01  維修側
      AND     L3430  ; 出右開夾位置01  操作側
      AND     L2230  ; 合流後掛框位置01進料側
      ANI     L3313  ; 出左開夾歸零要求
      ANI     L3413  ; 出右開夾歸零要求
      AND     Y0A01  ; All AxisServo On
      OUT     L280  ; 允許出料開爪一行程
4885  LD      SM400  ; Run On\
      MPS
      AND>    D1060 K4  ; 出料框架來源尺寸寬1=250
      MOV     K4 D1060
      MRD
      AND<    D1060 K1  ; 出料框架來源尺寸寬1=250
      MOV     K1 D1060
      MPP
      DECO    D1060 M180 K3  ; 0
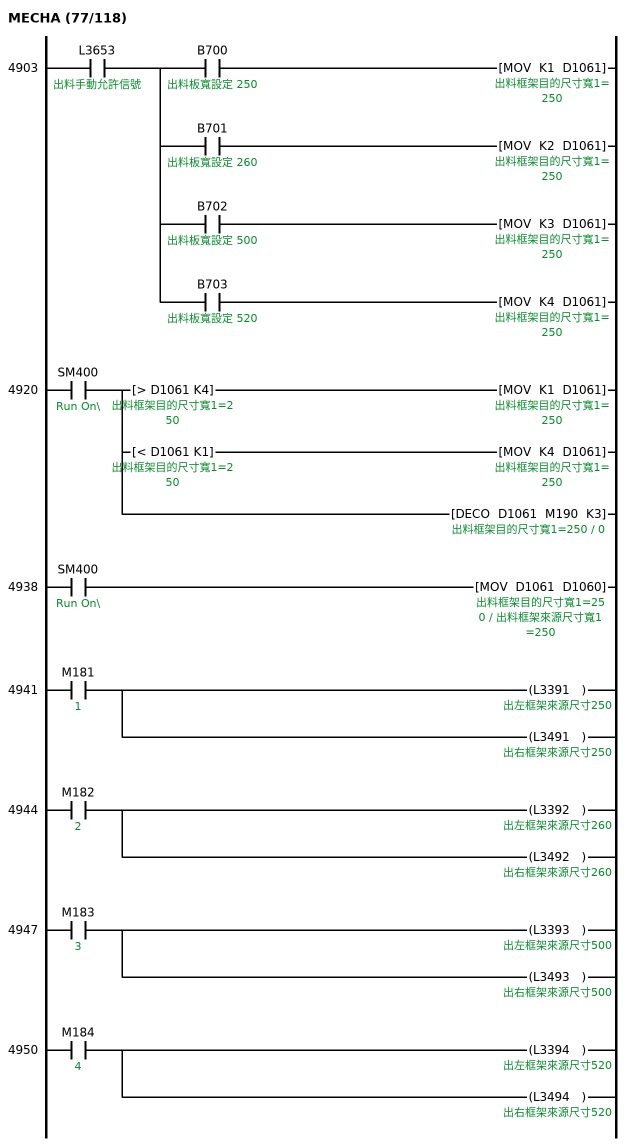
4903  LD      L3653  ; 出料手動允許信號
      MPS
      AND     B700  ; 出料板寬設定 250
      MOV     K1 D1061  ; 出料框架目的尺寸寬1=250
      MRD
      AND     B701  ; 出料板寬設定 260
      MOV     K2 D1061
      MRD
      AND     B702  ; 出料板寬設定 500
      MOV     K3 D1061
      MPP
      AND     B703  ; 出料板寬設定 520
      MOV     K4 D1061
4920  LD      SM400  ; Run On\
      MPS
      AND>    D1061 K4  ; 出料框架目的尺寸寬1=250
      MOV     K1 D1061
      MRD
      AND<    D1061 K1  ; 出料框架目的尺寸寬1=250
      MOV     K4 D1061
      MPP
      DECO    D1061 M190 K3  ; 0
4938  LD      SM400  ; Run On\
      MOV     D1061 D1060
4941  LD      M181  ; 1
      OUT     L3391  ; 出左框架來源尺寸250
      OUT     L3491  ; 出右框架來源尺寸250
4944  LD      M182  ; 2
      OUT     L3392  ; 出左框架來源尺寸260
      OUT     L3492  ; 出右框架來源尺寸260
4947  LD      M183  ; 3
      OUT     L3393  ; 出左框架來源尺寸500
      OUT     L3493  ; 出右框架來源尺寸500
4950  LD      M184  ; 4
      OUT     L3394  ; 出左框架來源尺寸520
      OUT     L3494  ; 出右框架來源尺寸520
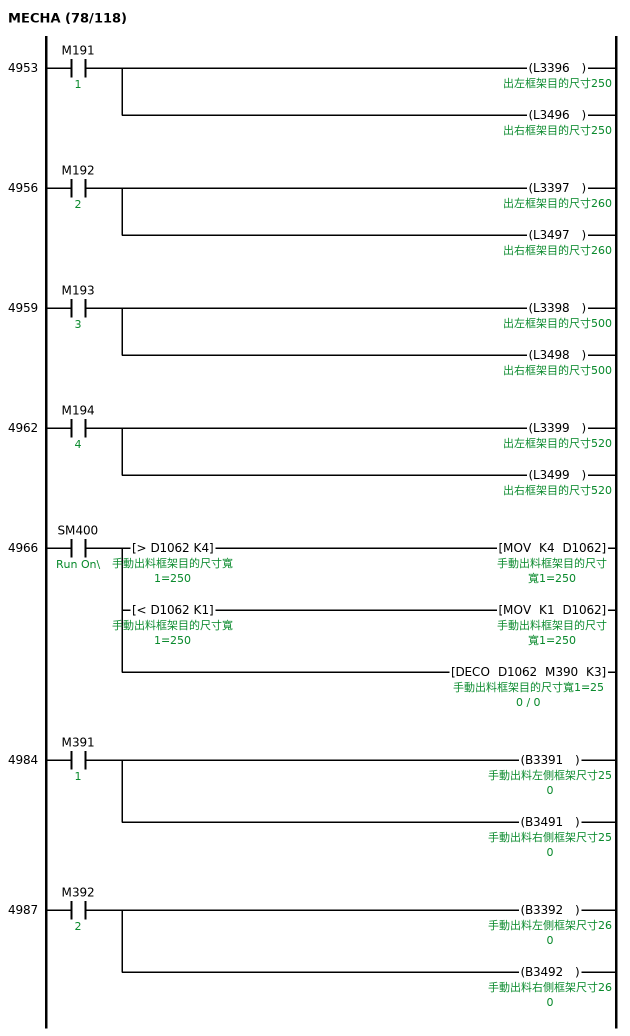
4953  LD      M191  ; 1
      OUT     L3396  ; 出左框架目的尺寸250
      OUT     L3496  ; 出右框架目的尺寸250
4956  LD      M192  ; 2
      OUT     L3397  ; 出左框架目的尺寸260
      OUT     L3497  ; 出右框架目的尺寸260
4959  LD      M193  ; 3
      OUT     L3398  ; 出左框架目的尺寸500
      OUT     L3498  ; 出右框架目的尺寸500
4962  LD      M194  ; 4
      OUT     L3399  ; 出左框架目的尺寸520
      OUT     L3499  ; 出右框架目的尺寸520
4966  LD      SM400  ; Run On\
      MPS
      AND>    D1062 K4  ; 手動出料框架目的尺寸寬1=250
      MOV     K4 D1062
      MRD
      AND<    D1062 K1  ; 手動出料框架目的尺寸寬1=250
      MOV     K1 D1062
      MPP
      DECO    D1062 M390 K3  ; 0
4984  LD      M391  ; 1
      OUT     B3391  ; 手動出料左側框架尺寸250
      OUT     B3491  ; 手動出料右側框架尺寸250
4987  LD      M392  ; 2
      OUT     B3392  ; 手動出料左側框架尺寸260
      OUT     B3492  ; 手動出料右側框架尺寸260
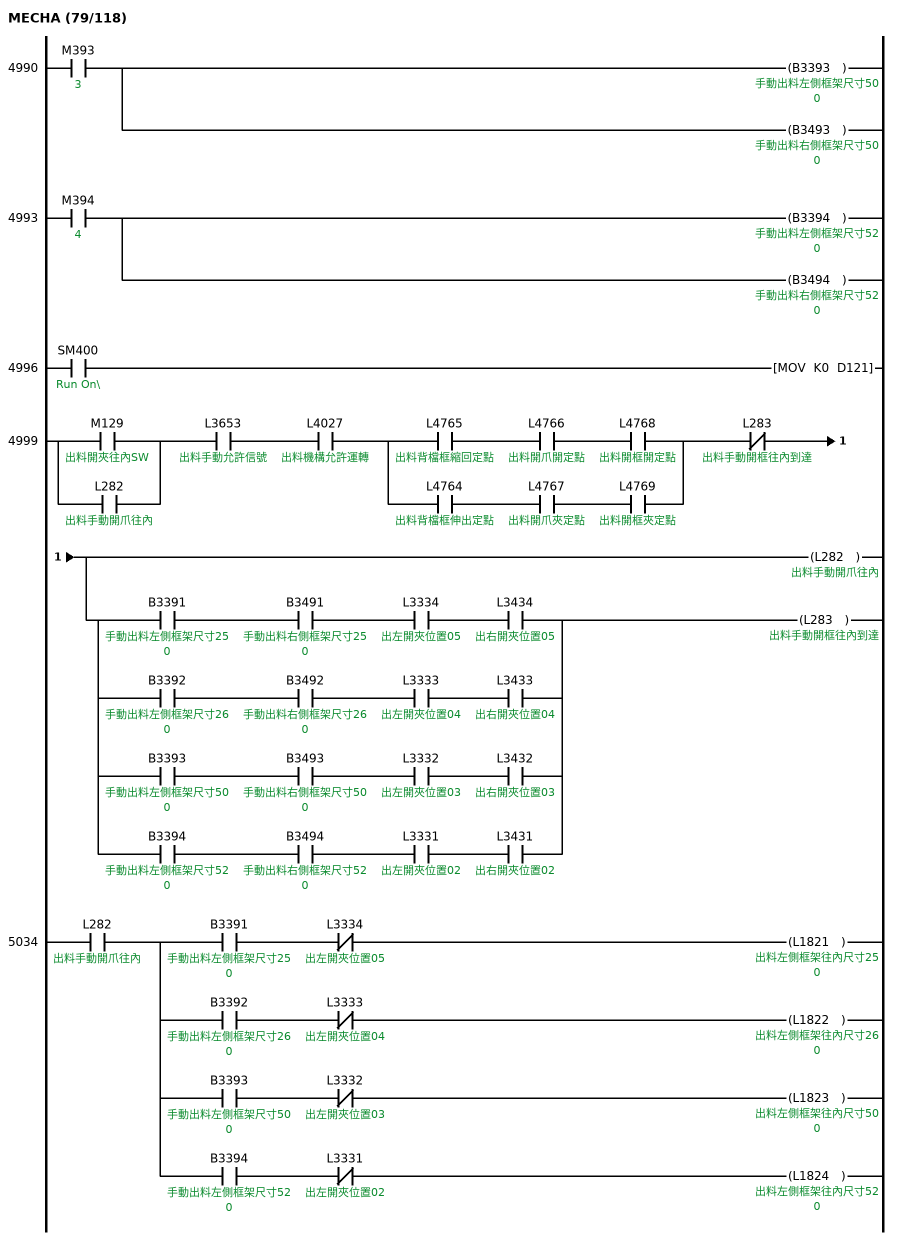
4990  LD      M393  ; 3
      OUT     B3393  ; 手動出料左側框架尺寸500
      OUT     B3493  ; 手動出料右側框架尺寸500
4993  LD      M394  ; 4
      OUT     B3394  ; 手動出料左側框架尺寸520
      OUT     B3494  ; 手動出料右側框架尺寸520
4996  LD      SM400  ; Run On\
      MOV     K0 D121
4999  LD      M129  ; 出料開夾往內SW
      OR      L282  ; 出料手動開爪往內
      AND     L3653  ; 出料手動允許信號
      AND     L4027  ; 出料機構允許運轉
      LD      L4765  ; 出料背檔框縮回定點
      AND     L4766  ; 出料開爪開定點
      AND     L4768  ; 出料開框開定點
      LD      L4764  ; 出料背檔框伸出定點
      AND     L4767  ; 出料開爪夾定點
      AND     L4769  ; 出料開框夾定點
      ORB
      ANB
      ANI     L283  ; 出料手動開框往內到達
      OUT     L282  ; 出料手動開爪往內
      LD      B3391  ; 手動出料左側框架尺寸250
      AND     B3491  ; 手動出料右側框架尺寸250
      AND     L3334  ; 出左開夾位置05
      AND     L3434  ; 出右開夾位置05
      LD      B3392  ; 手動出料左側框架尺寸260
      AND     B3492  ; 手動出料右側框架尺寸260
      AND     L3333  ; 出左開夾位置04
      AND     L3433  ; 出右開夾位置04
      ORB
      LD      B3393  ; 手動出料左側框架尺寸500
      AND     B3493  ; 手動出料右側框架尺寸500
      AND     L3332  ; 出左開夾位置03
      AND     L3432  ; 出右開夾位置03
      ORB
      LD      B3394  ; 手動出料左側框架尺寸520
      AND     B3494  ; 手動出料右側框架尺寸520
      AND     L3331  ; 出左開夾位置02
      AND     L3431  ; 出右開夾位置02
      ORB
      ANB
      OUT     L283  ; 出料手動開框往內到達
5034  LD      L282  ; 出料手動開爪往內
      MPS
      AND     B3391  ; 手動出料左側框架尺寸250
      ANI     L3334  ; 出左開夾位置05
      OUT     L1821  ; 出料左側框架往內尺寸250
      MRD
      AND     B3392  ; 手動出料左側框架尺寸260
      ANI     L3333  ; 出左開夾位置04
      OUT     L1822  ; 出料左側框架往內尺寸260
      MRD
      AND     B3393  ; 手動出料左側框架尺寸500
      ANI     L3332  ; 出左開夾位置03
      OUT     L1823  ; 出料左側框架往內尺寸500
      MPP
      AND     B3394  ; 手動出料左側框架尺寸520
      ANI     L3331  ; 出左開夾位置02
      OUT     L1824  ; 出料左側框架往內尺寸520
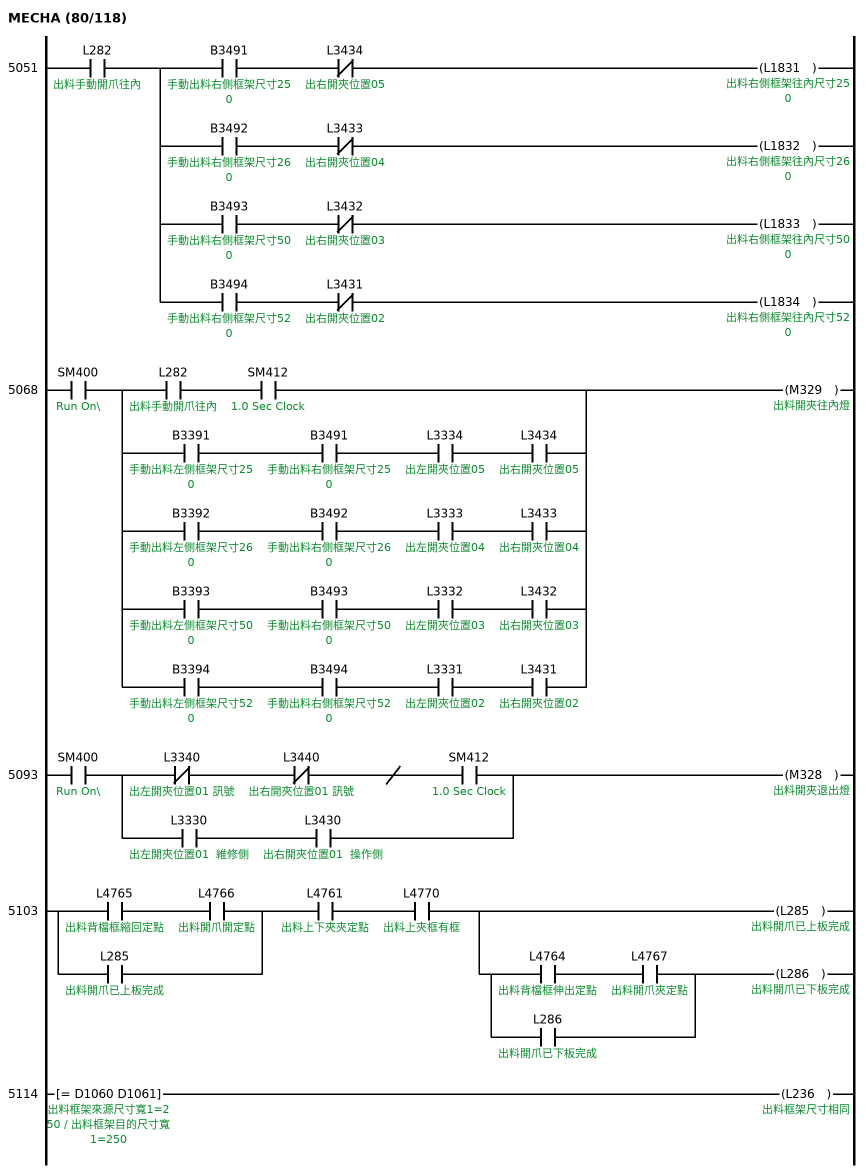
5051  LD      L282  ; 出料手動開爪往內
      MPS
      AND     B3491  ; 手動出料右側框架尺寸250
      ANI     L3434  ; 出右開夾位置05
      OUT     L1831  ; 出料右側框架往內尺寸250
      MRD
      AND     B3492  ; 手動出料右側框架尺寸260
      ANI     L3433  ; 出右開夾位置04
      OUT     L1832  ; 出料右側框架往內尺寸260
      MRD
      AND     B3493  ; 手動出料右側框架尺寸500
      ANI     L3432  ; 出右開夾位置03
      OUT     L1833  ; 出料右側框架往內尺寸500
      MPP
      AND     B3494  ; 手動出料右側框架尺寸520
      ANI     L3431  ; 出右開夾位置02
      OUT     L1834  ; 出料右側框架往內尺寸520
5068  LD      SM400  ; Run On\
      LD      L282  ; 出料手動開爪往內
      AND     SM412  ; 1.0 Sec Clock
      LD      B3391  ; 手動出料左側框架尺寸250
      AND     B3491  ; 手動出料右側框架尺寸250
      AND     L3334  ; 出左開夾位置05
      AND     L3434  ; 出右開夾位置05
      ORB
      LD      B3392  ; 手動出料左側框架尺寸260
      AND     B3492  ; 手動出料右側框架尺寸260
      AND     L3333  ; 出左開夾位置04
      AND     L3433  ; 出右開夾位置04
      ORB
      LD      B3393  ; 手動出料左側框架尺寸500
      AND     B3493  ; 手動出料右側框架尺寸500
      AND     L3332  ; 出左開夾位置03
      AND     L3432  ; 出右開夾位置03
      ORB
      LD      B3394  ; 手動出料左側框架尺寸520
      AND     B3494  ; 手動出料右側框架尺寸520
      AND     L3331  ; 出左開夾位置02
      AND     L3431  ; 出右開夾位置02
      ORB
      ANB
      OUT     M329  ; 出料開夾往內燈
5093  LD      SM400  ; Run On\
      LDI     L3340  ; 出左開夾位置01 訊號
      ANI     L3440  ; 出右開夾位置01 訊號
      INV
      AND     SM412  ; 1.0 Sec Clock
      LD      L3330  ; 出左開夾位置01  維修側
      AND     L3430  ; 出右開夾位置01  操作側
      ORB
      ANB
      OUT     M328  ; 出料開夾退出燈
5103  LD      L4765  ; 出料背檔框縮回定點
      AND     L4766  ; 出料開爪開定點
      OR      L285  ; 出料開爪已上板完成
      AND     L4761  ; 出料上下夾夾定點
      AND     L4770  ; 出料上夾框有框
      OUT     L285  ; 出料開爪已上板完成
      LD      L4764  ; 出料背檔框伸出定點
      AND     L4767  ; 出料開爪夾定點
      OR      L286  ; 出料開爪已下板完成
      ANB
      OUT     L286  ; 出料開爪已下板完成
5114  LD=     D1060 D1061  ; 出料框架來源尺寸寬1=250 / 出料框架目的尺寸寬1=250
      OUT     L236  ; 出料框架尺寸相同
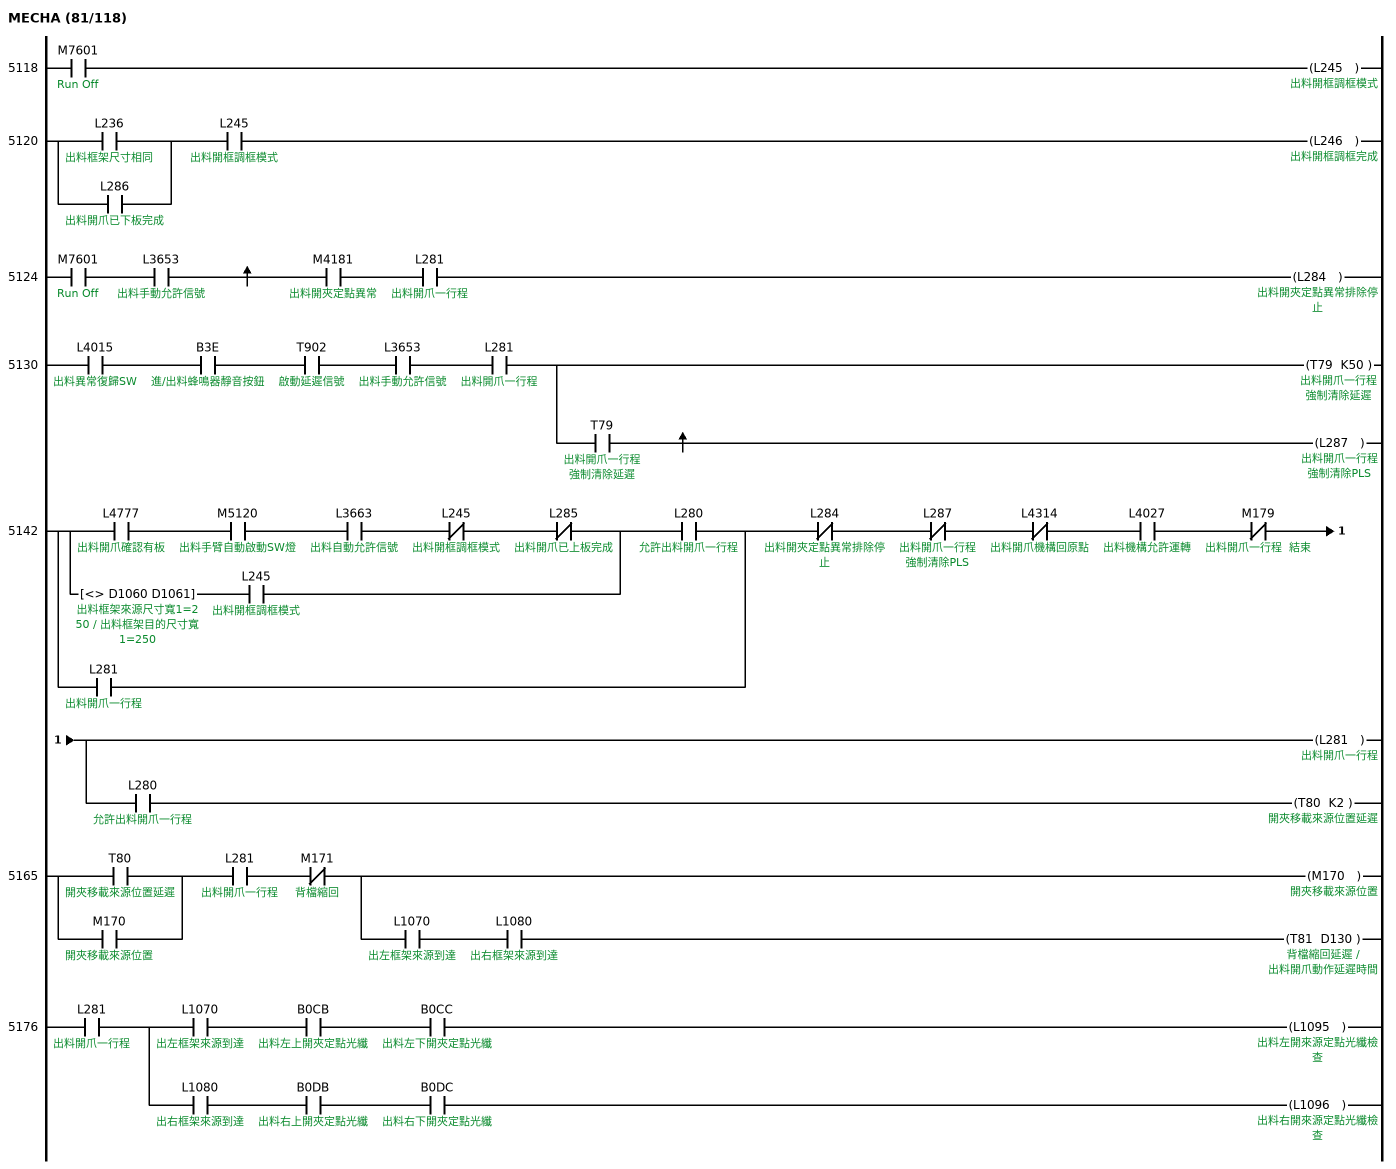
5118  LD      M7601  ; Run Off
      OUT     L245  ; 出料開框調框模式
5120  LD      L236  ; 出料框架尺寸相同
      OR      L286  ; 出料開爪已下板完成
      AND     L245  ; 出料開框調框模式
      OUT     L246  ; 出料開框調框完成
5124  LD      M7601  ; Run Off
      AND     L3653  ; 出料手動允許信號
      MEP
      AND     M4181  ; 出料開夾定點異常
      AND     L281  ; 出料開爪一行程
      OUT     L284  ; 出料開夾定點異常排除停止
5130  LD      L4015  ; 出料異常復歸SW
      AND     B3E  ; 進/出料蜂鳴器靜音按鈕
      AND     T902  ; 啟動延遲信號
      AND     L3653  ; 出料手動允許信號
      AND     L281  ; 出料開爪一行程
      OUT     T79 K50  ; 出料開爪一行程  強制清除延遲
      AND     T79  ; 出料開爪一行程  強制清除延遲
      MEP
      OUT     L287  ; 出料開爪一行程  強制清除PLS
5142  LD      L4777  ; 出料開爪確認有板
      AND     M5120  ; 出料手臂自動啟動SW燈
      AND     L3663  ; 出料自動允許信號
      ANI     L245  ; 出料開框調框模式
      ANI     L285  ; 出料開爪已上板完成
      LD<>    D1060 D1061  ; 出料框架來源尺寸寬1=250 / 出料框架目的尺寸寬1=250
      AND     L245  ; 出料開框調框模式
      ORB
      AND     L280  ; 允許出料開爪一行程
      OR      L281  ; 出料開爪一行程
      ANI     L284  ; 出料開夾定點異常排除停止
      ANI     L287  ; 出料開爪一行程  強制清除PLS
      ANI     L4314  ; 出料開爪機構回原點
      AND     L4027  ; 出料機構允許運轉
      ANI     M179  ; 出料開爪一行程  結束
      OUT     L281  ; 出料開爪一行程
      AND     L280  ; 允許出料開爪一行程
      OUT     T80 K2  ; 開夾移載來源位置延遲
5165  LD      T80  ; 開夾移載來源位置延遲
      OR      M170  ; 開夾移載來源位置
      AND     L281  ; 出料開爪一行程
      ANI     M171  ; 背檔縮回
      OUT     M170  ; 開夾移載來源位置
      AND     L1070  ; 出左框架來源到達
      AND     L1080  ; 出右框架來源到達
      OUT     T81 D130  ; 背檔縮回延遲 / 出料開爪動作延遲時間
5176  LD      L281  ; 出料開爪一行程
      MPS
      AND     L1070  ; 出左框架來源到達
      AND     B0CB  ; 出料左上開夾定點光纖
      AND     B0CC  ; 出料左下開夾定點光纖
      OUT     L1095  ; 出料左開來源定點光纖檢查
      MPP
      AND     L1080  ; 出右框架來源到達
      AND     B0DB  ; 出料右上開夾定點光纖
      AND     B0DC  ; 出料右下開夾定點光纖
      OUT     L1096  ; 出料右開來源定點光纖檢查
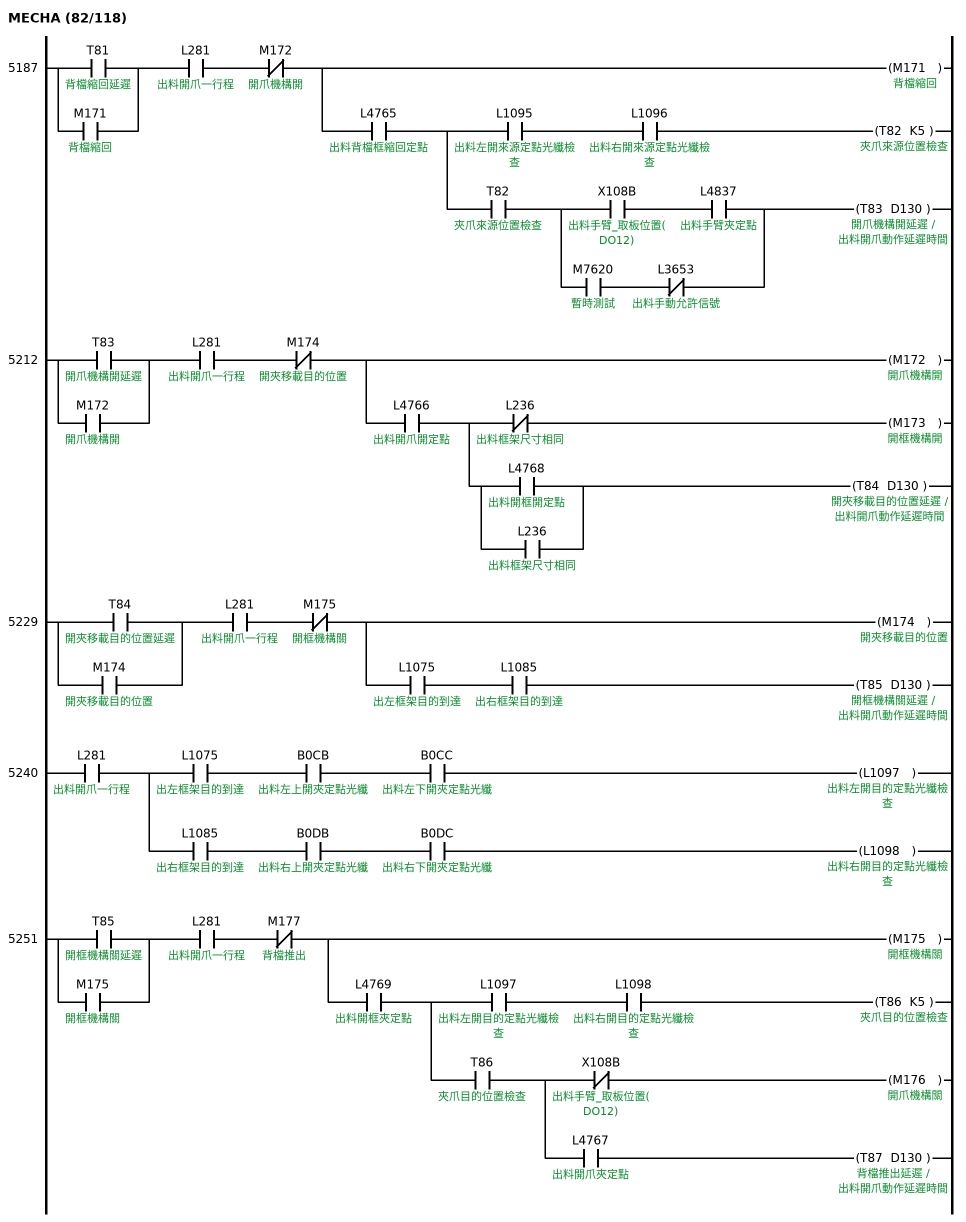
5187  LD      T81  ; 背檔縮回延遲
      OR      M171  ; 背檔縮回
      AND     L281  ; 出料開爪一行程
      ANI     M172  ; 開爪機構開
      OUT     M171  ; 背檔縮回
      AND     L4765  ; 出料背檔框縮回定點
      MPS
      AND     L1095  ; 出料左開來源定點光纖檢查
      AND     L1096  ; 出料右開來源定點光纖檢查
      OUT     T82 K5  ; 夾爪來源位置檢查
      MPP
      AND     T82  ; 夾爪來源位置檢查
      LD      X108B  ; 出料手臂_取板位置(DO12)
      AND     L4837  ; 出料手臂夾定點
      LD      M7620  ; 暫時測試
      ANI     L3653  ; 出料手動允許信號
      ORB
      ANB
      OUT     T83 D130  ; 開爪機構開延遲 / 出料開爪動作延遲時間
5212  LD      T83  ; 開爪機構開延遲
      OR      M172  ; 開爪機構開
      AND     L281  ; 出料開爪一行程
      ANI     M174  ; 開夾移載目的位置
      OUT     M172  ; 開爪機構開
      AND     L4766  ; 出料開爪開定點
      MPS
      ANI     L236  ; 出料框架尺寸相同
      OUT     M173  ; 開框機構開
      MPP
      LD      L4768  ; 出料開框開定點
      OR      L236  ; 出料框架尺寸相同
      ANB
      OUT     T84 D130  ; 開夾移載目的位置延遲 / 出料開爪動作延遲時間
5229  LD      T84  ; 開夾移載目的位置延遲
      OR      M174  ; 開夾移載目的位置
      AND     L281  ; 出料開爪一行程
      ANI     M175  ; 開框機構關
      OUT     M174  ; 開夾移載目的位置
      AND     L1075  ; 出左框架目的到達
      AND     L1085  ; 出右框架目的到達
      OUT     T85 D130  ; 開框機構關延遲 / 出料開爪動作延遲時間
5240  LD      L281  ; 出料開爪一行程
      MPS
      AND     L1075  ; 出左框架目的到達
      AND     B0CB  ; 出料左上開夾定點光纖
      AND     B0CC  ; 出料左下開夾定點光纖
      OUT     L1097  ; 出料左開目的定點光纖檢查
      MPP
      AND     L1085  ; 出右框架目的到達
      AND     B0DB  ; 出料右上開夾定點光纖
      AND     B0DC  ; 出料右下開夾定點光纖
      OUT     L1098  ; 出料右開目的定點光纖檢查
5251  LD      T85  ; 開框機構關延遲
      OR      M175  ; 開框機構關
      AND     L281  ; 出料開爪一行程
      ANI     M177  ; 背檔推出
      OUT     M175  ; 開框機構關
      AND     L4769  ; 出料開框夾定點
      MPS
      AND     L1097  ; 出料左開目的定點光纖檢查
      AND     L1098  ; 出料右開目的定點光纖檢查
      OUT     T86 K5  ; 夾爪目的位置檢查
      MPP
      AND     T86  ; 夾爪目的位置檢查
      MPS
      ANI     X108B  ; 出料手臂_取板位置(DO12)
      OUT     M176  ; 開爪機構關
      MPP
      AND     L4767  ; 出料開爪夾定點
      OUT     T87 D130  ; 背檔推出延遲 / 出料開爪動作延遲時間
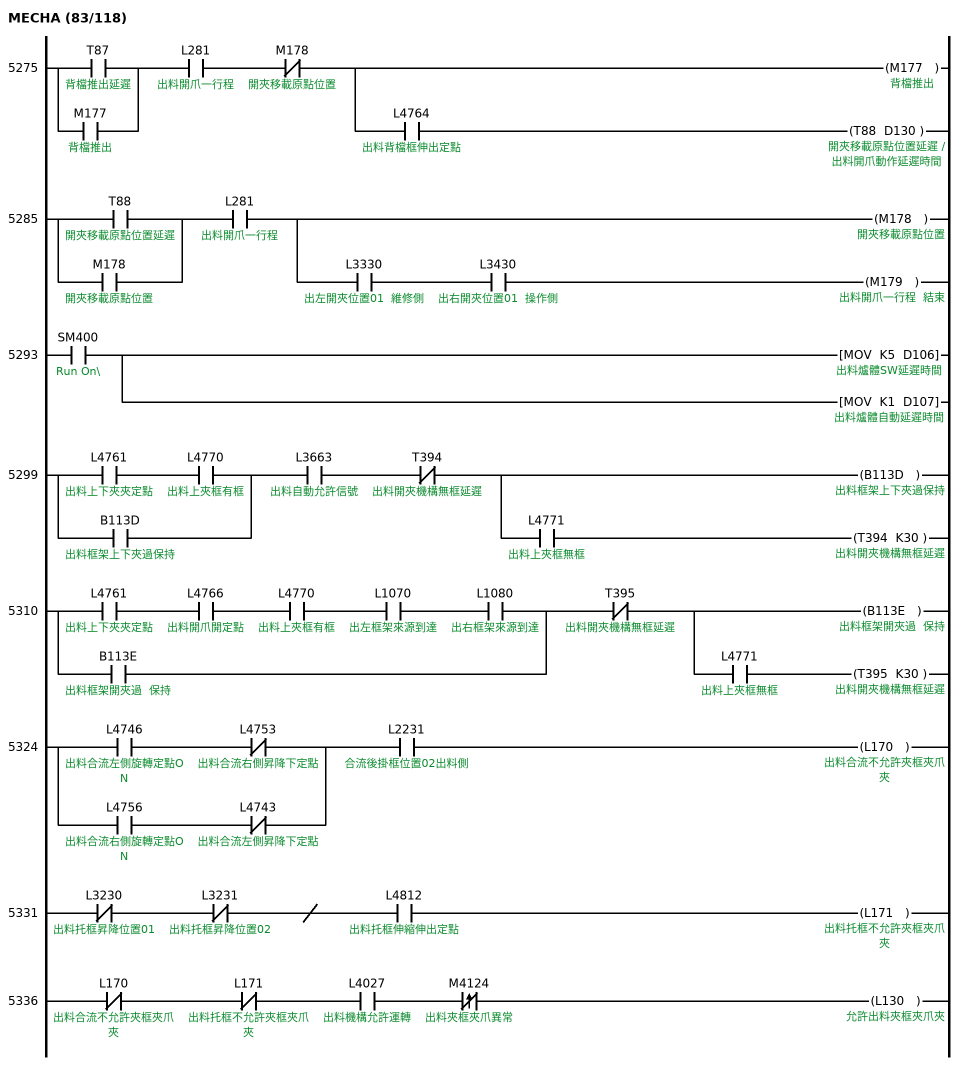
5275  LD      T87  ; 背檔推出延遲
      OR      M177  ; 背檔推出
      AND     L281  ; 出料開爪一行程
      ANI     M178  ; 開夾移載原點位置
      OUT     M177  ; 背檔推出
      AND     L4764  ; 出料背檔框伸出定點
      OUT     T88 D130  ; 開夾移載原點位置延遲 / 出料開爪動作延遲時間
5285  LD      T88  ; 開夾移載原點位置延遲
      OR      M178  ; 開夾移載原點位置
      AND     L281  ; 出料開爪一行程
      OUT     M178  ; 開夾移載原點位置
      AND     L3330  ; 出左開夾位置01  維修側
      AND     L3430  ; 出右開夾位置01  操作側
      OUT     M179  ; 出料開爪一行程  結束
5293  LD      SM400  ; Run On\
      MOV     K5 D106  ; 出料爐體SW延遲時間
      MOV     K1 D107  ; 出料爐體自動延遲時間
5299  LD      L4761  ; 出料上下夾夾定點
      AND     L4770  ; 出料上夾框有框
      OR      B113D  ; 出料框架上下夾過保持
      AND     L3663  ; 出料自動允許信號
      ANI     T394  ; 出料開夾機構無框延遲
      OUT     B113D  ; 出料框架上下夾過保持
      AND     L4771  ; 出料上夾框無框
      OUT     T394 K30  ; 出料開夾機構無框延遲
5310  LD      L4761  ; 出料上下夾夾定點
      AND     L4766  ; 出料開爪開定點
      AND     L4770  ; 出料上夾框有框
      AND     L1070  ; 出左框架來源到達
      AND     L1080  ; 出右框架來源到達
      OR      B113E  ; 出料框架開夾過  保持
      ANI     T395  ; 出料開夾機構無框延遲
      OUT     B113E  ; 出料框架開夾過  保持
      AND     L4771  ; 出料上夾框無框
      OUT     T395 K30  ; 出料開夾機構無框延遲
5324  LD      L4746  ; 出料合流左側旋轉定點ON
      ANI     L4753  ; 出料合流右側昇降下定點
      LD      L4756  ; 出料合流右側旋轉定點ON
      ANI     L4743  ; 出料合流左側昇降下定點
      ORB
      AND     L2231  ; 合流後掛框位置02出料側
      OUT     L170  ; 出料合流不允許夾框夾爪夾
5331  LDI     L3230  ; 出料托框昇降位置01
      ANI     L3231  ; 出料托框昇降位置02
      INV
      AND     L4812  ; 出料托框伸縮伸出定點
      OUT     L171  ; 出料托框不允許夾框夾爪夾
5336  LDI     L170  ; 出料合流不允許夾框夾爪夾
      ANI     L171  ; 出料托框不允許夾框夾爪夾
      AND     L4027  ; 出料機構允許運轉
      ANDPI   M4124  ; 出料夾框夾爪異常
      OUT     L130  ; 允許出料夾框夾爪夾
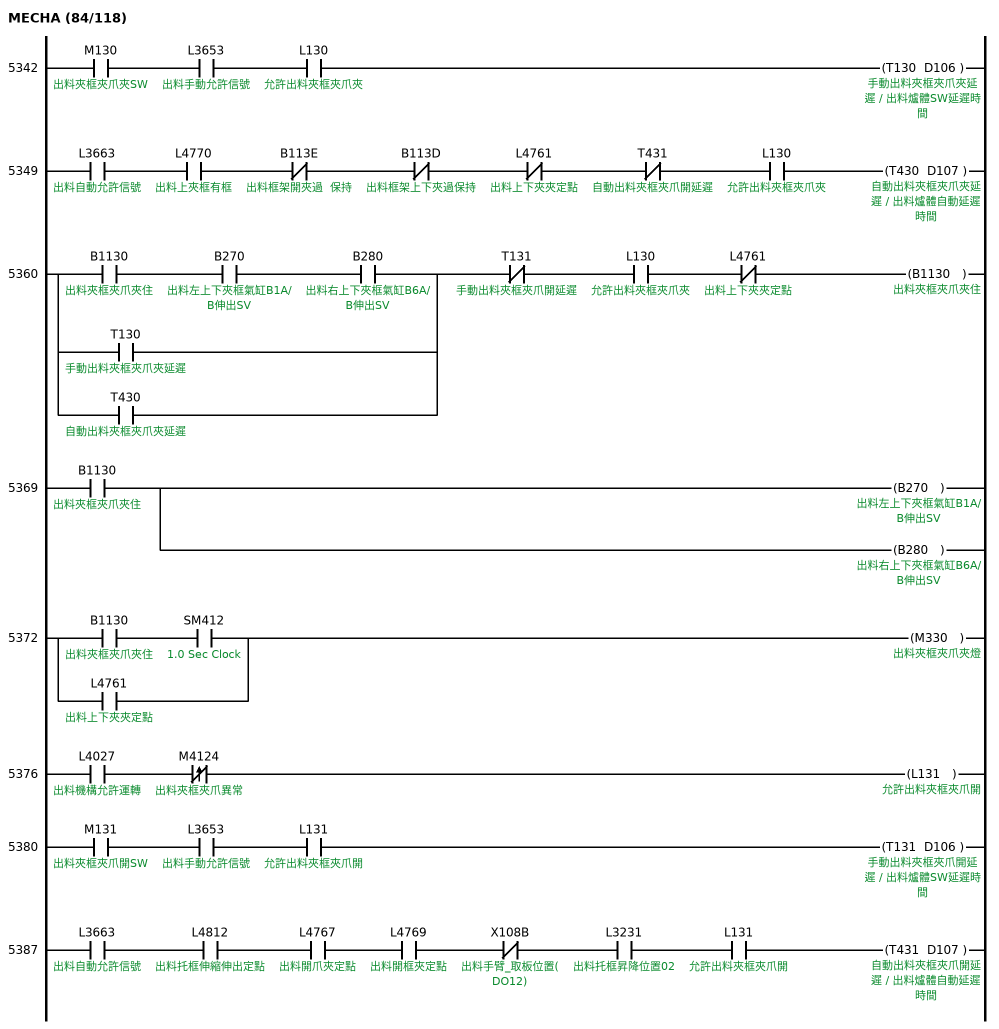
5342  LD      M130  ; 出料夾框夾爪夾SW
      AND     L3653  ; 出料手動允許信號
      AND     L130  ; 允許出料夾框夾爪夾
      OUT     T130 D106  ; 手動出料夾框夾爪夾延遲 / 出料爐體SW延遲時間
5349  LD      L3663  ; 出料自動允許信號
      AND     L4770  ; 出料上夾框有框
      ANI     B113E  ; 出料框架開夾過  保持
      ANI     B113D  ; 出料框架上下夾過保持
      ANI     L4761  ; 出料上下夾夾定點
      ANI     T431  ; 自動出料夾框夾爪開延遲
      AND     L130  ; 允許出料夾框夾爪夾
      OUT     T430 D107  ; 自動出料夾框夾爪夾延遲 / 出料爐體自動延遲時間
5360  LD      B1130  ; 出料夾框夾爪夾住
      AND     B270  ; 出料左上下夾框氣缸B1A/B伸出SV
      AND     B280  ; 出料右上下夾框氣缸B6A/B伸出SV
      OR      T130  ; 手動出料夾框夾爪夾延遲
      OR      T430  ; 自動出料夾框夾爪夾延遲
      ANI     T131  ; 手動出料夾框夾爪開延遲
      AND     L130  ; 允許出料夾框夾爪夾
      ANI     L4761  ; 出料上下夾夾定點
      OUT     B1130  ; 出料夾框夾爪夾住
5369  LD      B1130  ; 出料夾框夾爪夾住
      OUT     B270  ; 出料左上下夾框氣缸B1A/B伸出SV
      OUT     B280  ; 出料右上下夾框氣缸B6A/B伸出SV
5372  LD      B1130  ; 出料夾框夾爪夾住
      AND     SM412  ; 1.0 Sec Clock
      OR      L4761  ; 出料上下夾夾定點
      OUT     M330  ; 出料夾框夾爪夾燈
5376  LD      L4027  ; 出料機構允許運轉
      ANDPI   M4124  ; 出料夾框夾爪異常
      OUT     L131  ; 允許出料夾框夾爪開
5380  LD      M131  ; 出料夾框夾爪開SW
      AND     L3653  ; 出料手動允許信號
      AND     L131  ; 允許出料夾框夾爪開
      OUT     T131 D106  ; 手動出料夾框夾爪開延遲 / 出料爐體SW延遲時間
5387  LD      L3663  ; 出料自動允許信號
      AND     L4812  ; 出料托框伸縮伸出定點
      AND     L4767  ; 出料開爪夾定點
      AND     L4769  ; 出料開框夾定點
      ANI     X108B  ; 出料手臂_取板位置(DO12)
      AND     L3231  ; 出料托框昇降位置02
      AND     L131  ; 允許出料夾框夾爪開
      OUT     T431 D107  ; 自動出料夾框夾爪開延遲 / 出料爐體自動延遲時間
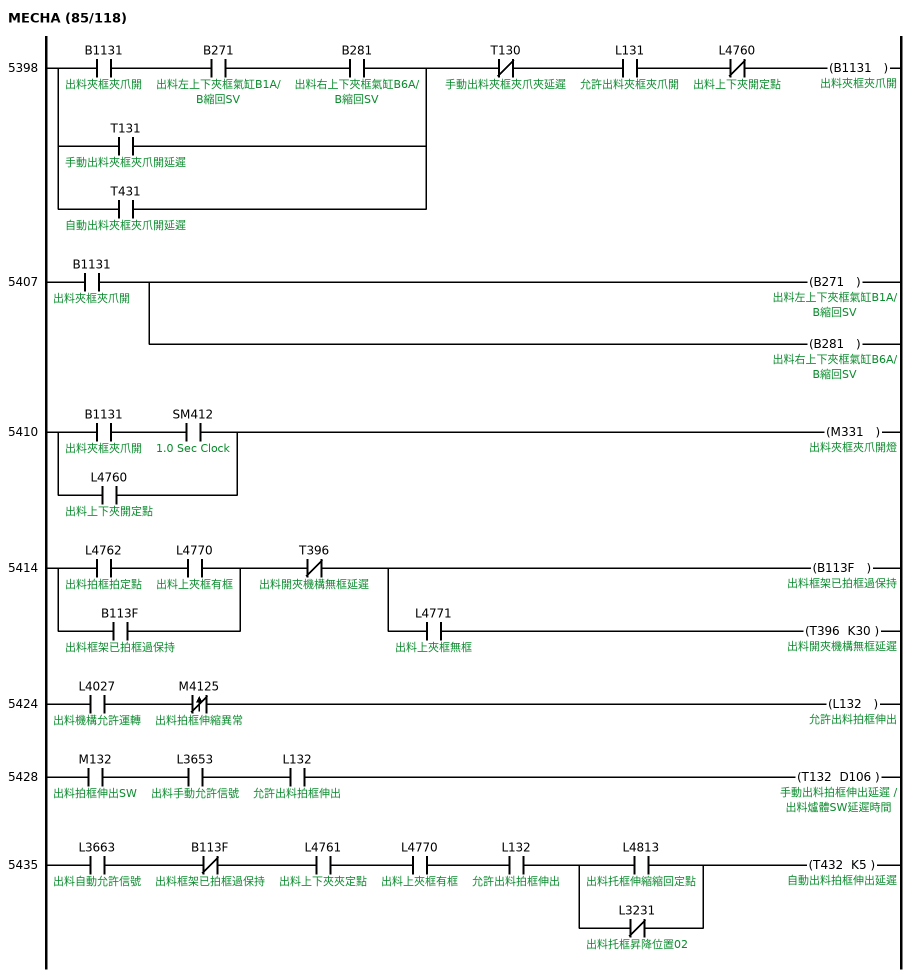
5398  LD      B1131  ; 出料夾框夾爪開
      AND     B271  ; 出料左上下夾框氣缸B1A/B縮回SV
      AND     B281  ; 出料右上下夾框氣缸B6A/B縮回SV
      OR      T131  ; 手動出料夾框夾爪開延遲
      OR      T431  ; 自動出料夾框夾爪開延遲
      ANI     T130  ; 手動出料夾框夾爪夾延遲
      AND     L131  ; 允許出料夾框夾爪開
      ANI     L4760  ; 出料上下夾開定點
      OUT     B1131  ; 出料夾框夾爪開
5407  LD      B1131  ; 出料夾框夾爪開
      OUT     B271  ; 出料左上下夾框氣缸B1A/B縮回SV
      OUT     B281  ; 出料右上下夾框氣缸B6A/B縮回SV
5410  LD      B1131  ; 出料夾框夾爪開
      AND     SM412  ; 1.0 Sec Clock
      OR      L4760  ; 出料上下夾開定點
      OUT     M331  ; 出料夾框夾爪開燈
5414  LD      L4762  ; 出料拍框拍定點
      AND     L4770  ; 出料上夾框有框
      OR      B113F  ; 出料框架已拍框過保持
      ANI     T396  ; 出料開夾機構無框延遲
      OUT     B113F  ; 出料框架已拍框過保持
      AND     L4771  ; 出料上夾框無框
      OUT     T396 K30  ; 出料開夾機構無框延遲
5424  LD      L4027  ; 出料機構允許運轉
      ANDPI   M4125  ; 出料拍框伸縮異常
      OUT     L132  ; 允許出料拍框伸出
5428  LD      M132  ; 出料拍框伸出SW
      AND     L3653  ; 出料手動允許信號
      AND     L132  ; 允許出料拍框伸出
      OUT     T132 D106  ; 手動出料拍框伸出延遲 / 出料爐體SW延遲時間
5435  LD      L3663  ; 出料自動允許信號
      ANI     B113F  ; 出料框架已拍框過保持
      AND     L4761  ; 出料上下夾夾定點
      AND     L4770  ; 出料上夾框有框
      AND     L132  ; 允許出料拍框伸出
      LD      L4813  ; 出料托框伸縮縮回定點
      ORI     L3231  ; 出料托框昇降位置02
      ANB
      OUT     T432 K5  ; 自動出料拍框伸出延遲
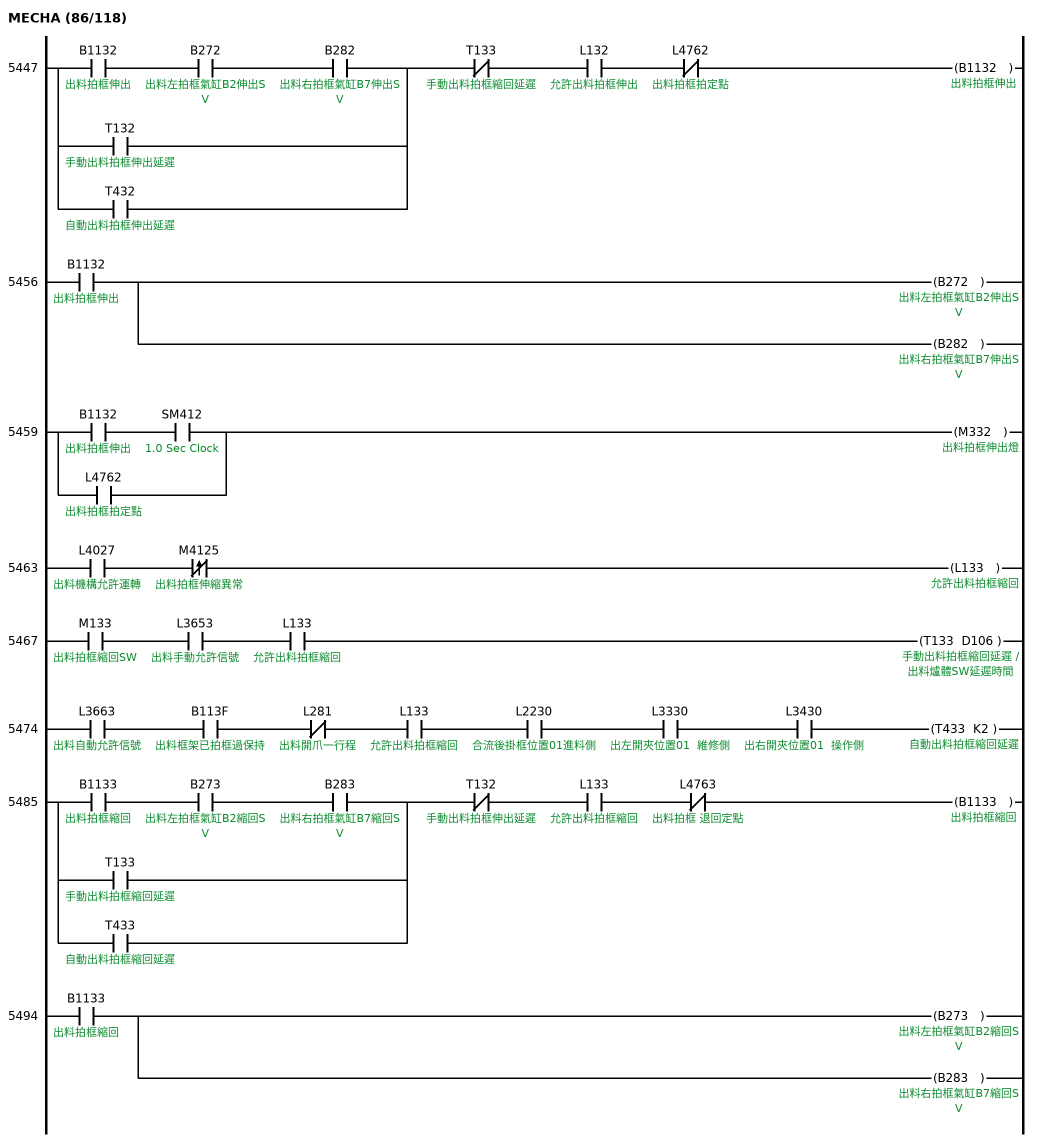
5447  LD      B1132  ; 出料拍框伸出
      AND     B272  ; 出料左拍框氣缸B2伸出SV
      AND     B282  ; 出料右拍框氣缸B7伸出SV
      OR      T132  ; 手動出料拍框伸出延遲
      OR      T432  ; 自動出料拍框伸出延遲
      ANI     T133  ; 手動出料拍框縮回延遲
      AND     L132  ; 允許出料拍框伸出
      ANI     L4762  ; 出料拍框拍定點
      OUT     B1132  ; 出料拍框伸出
5456  LD      B1132  ; 出料拍框伸出
      OUT     B272  ; 出料左拍框氣缸B2伸出SV
      OUT     B282  ; 出料右拍框氣缸B7伸出SV
5459  LD      B1132  ; 出料拍框伸出
      AND     SM412  ; 1.0 Sec Clock
      OR      L4762  ; 出料拍框拍定點
      OUT     M332  ; 出料拍框伸出燈
5463  LD      L4027  ; 出料機構允許運轉
      ANDPI   M4125  ; 出料拍框伸縮異常
      OUT     L133  ; 允許出料拍框縮回
5467  LD      M133  ; 出料拍框縮回SW
      AND     L3653  ; 出料手動允許信號
      AND     L133  ; 允許出料拍框縮回
      OUT     T133 D106  ; 手動出料拍框縮回延遲 / 出料爐體SW延遲時間
5474  LD      L3663  ; 出料自動允許信號
      AND     B113F  ; 出料框架已拍框過保持
      ANI     L281  ; 出料開爪一行程
      AND     L133  ; 允許出料拍框縮回
      AND     L2230  ; 合流後掛框位置01進料側
      AND     L3330  ; 出左開夾位置01  維修側
      AND     L3430  ; 出右開夾位置01  操作側
      OUT     T433 K2  ; 自動出料拍框縮回延遲
5485  LD      B1133  ; 出料拍框縮回
      AND     B273  ; 出料左拍框氣缸B2縮回SV
      AND     B283  ; 出料右拍框氣缸B7縮回SV
      OR      T133  ; 手動出料拍框縮回延遲
      OR      T433  ; 自動出料拍框縮回延遲
      ANI     T132  ; 手動出料拍框伸出延遲
      AND     L133  ; 允許出料拍框縮回
      ANI     L4763  ; 出料拍框 退回定點
      OUT     B1133  ; 出料拍框縮回
5494  LD      B1133  ; 出料拍框縮回
      OUT     B273  ; 出料左拍框氣缸B2縮回SV
      OUT     B283  ; 出料右拍框氣缸B7縮回SV
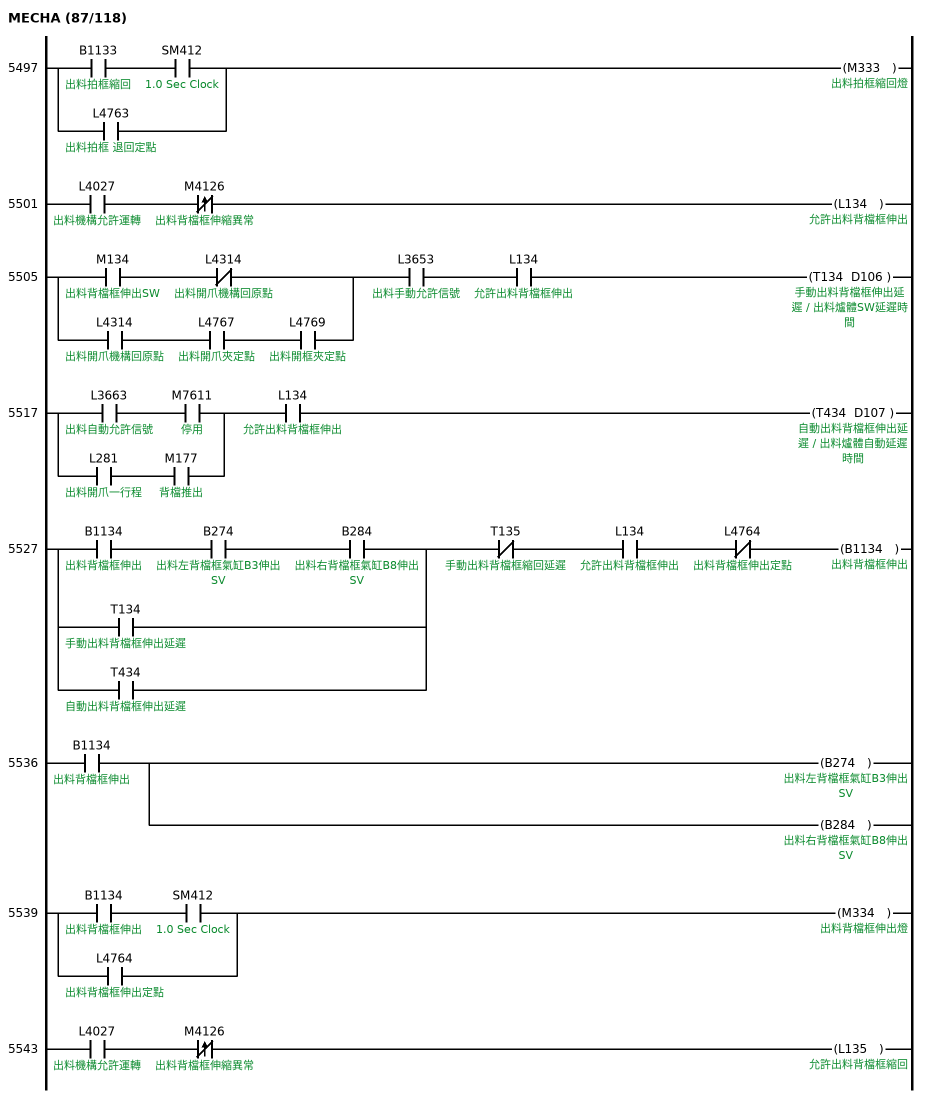
5497  LD      B1133  ; 出料拍框縮回
      AND     SM412  ; 1.0 Sec Clock
      OR      L4763  ; 出料拍框 退回定點
      OUT     M333  ; 出料拍框縮回燈
5501  LD      L4027  ; 出料機構允許運轉
      ANDPI   M4126  ; 出料背檔框伸縮異常
      OUT     L134  ; 允許出料背檔框伸出
5505  LD      M134  ; 出料背檔框伸出SW
      ANI     L4314  ; 出料開爪機構回原點
      LD      L4314  ; 出料開爪機構回原點
      AND     L4767  ; 出料開爪夾定點
      AND     L4769  ; 出料開框夾定點
      ORB
      AND     L3653  ; 出料手動允許信號
      AND     L134  ; 允許出料背檔框伸出
      OUT     T134 D106  ; 手動出料背檔框伸出延遲 / 出料爐體SW延遲時間
5517  LD      L3663  ; 出料自動允許信號
      AND     M7611  ; 停用
      LD      L281  ; 出料開爪一行程
      AND     M177  ; 背檔推出
      ORB
      AND     L134  ; 允許出料背檔框伸出
      OUT     T434 D107  ; 自動出料背檔框伸出延遲 / 出料爐體自動延遲時間
5527  LD      B1134  ; 出料背檔框伸出
      AND     B274  ; 出料左背檔框氣缸B3伸出SV
      AND     B284  ; 出料右背檔框氣缸B8伸出SV
      OR      T134  ; 手動出料背檔框伸出延遲
      OR      T434  ; 自動出料背檔框伸出延遲
      ANI     T135  ; 手動出料背檔框縮回延遲
      AND     L134  ; 允許出料背檔框伸出
      ANI     L4764  ; 出料背檔框伸出定點
      OUT     B1134  ; 出料背檔框伸出
5536  LD      B1134  ; 出料背檔框伸出
      OUT     B274  ; 出料左背檔框氣缸B3伸出SV
      OUT     B284  ; 出料右背檔框氣缸B8伸出SV
5539  LD      B1134  ; 出料背檔框伸出
      AND     SM412  ; 1.0 Sec Clock
      OR      L4764  ; 出料背檔框伸出定點
      OUT     M334  ; 出料背檔框伸出燈
5543  LD      L4027  ; 出料機構允許運轉
      ANDPI   M4126  ; 出料背檔框伸縮異常
      OUT     L135  ; 允許出料背檔框縮回
